KUKA KRL program: MyProgram_015().src

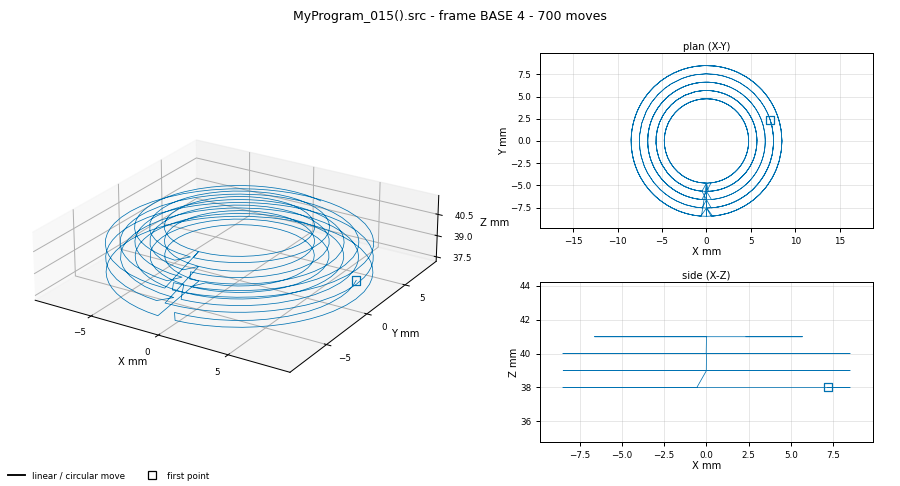
[picture p0: tool path of MyProgram_015().src in frame BASE 4, 700 of 700 moves have a stored position in this frame; points joined in program order, loops and branches not executed]
&ACCESS RVP
&REL 1
&PARAM TEMPLATE = C:\KRC\Roboter\Template\vorgabe
&PARAM EDITMASK = *
DEF MyProgram_015()
; ---- Setting reference (Base) ----
$BASE = BASE_DATA[4]

; --------------------------
; ---- Setting tool (TCP) ----
$TOOL = TOOL_DATA[3]
; --------------------------

$VEL.CP = VEL_APROX_PRINT
Startdeposition()
$VEL.CP = VEL_PRINT
LIN {X 7.1653,Y 2.4052,Z 38,A -2.3243,B 0,C 0,E1 0.1598,E2 90.0714} C_DIS
LIN {X 7.3844,Y 1.6056,Z 38,A -2.3508,B 0,C 0,E1 0.1598,E2 90.0719} C_DIS
LIN {X 7.5274,Y 0.6858,Z 38,A -2.3849,B 0,C 0,E1 0.1598,E2 90.0719} C_DIS
LIN {X 7.5543,Y -0.2016,Z 38,A -2.4217,B 0,C 0,E1 0.1598,E2 90.0719} C_DIS
LIN {X 7.4214,Y -1.405,Z 38,A -2.4775,B 0,C 0,E1 0.1598,E2 90.0714} C_DIS
LIN {X 7.2331,Y -2.1884,Z 38,A -2.5182,B 0,C 0,E1 0.1598,E2 90.0717} C_DIS
LIN {X 6.879,Y -3.1316,Z 38,A -2.5714,B 0,C 0,E1 0.1598,E2 90.0717} C_DIS
LIN {X 6.1912,Y -4.3324,Z 38,A -2.6476,B 0,C 0,E1 0.1598,E2 90.0712} C_DIS
LIN {X 5.3371,Y -5.3523,Z 38,A -2.7227,B 0,C 0,E1 0.1598,E2 90.0714} C_DIS
LIN {X 4.6683,Y -5.9424,Z 38,A -2.7727,B 0,C 0,E1 0.1598,E2 90.0717} C_DIS
LIN {X 3.7573,Y -6.5524,Z 38,A -2.8321,B 0,C 0,E1 0.1598,E2 90.0717} C_DIS
LIN {X 2.7191,Y -7.0514,Z 38,A -2.8915,B 0,C 0,E1 0.1598,E2 90.0717} C_DIS
LIN {X 1.7846,Y -7.3382,Z 38,A -2.9381,B 0,C 0,E1 0.1598,E2 90.0717} C_DIS
LIN {X 1.0166,Y -7.4849,Z 38,A -2.9725,B 0,C 0,E1 0.1598,E2 90.0717} C_DIS
LIN {X 0.0417,Y -7.5527,Z 38,A -3.0111,B 0,C 0,E1 0.1598,E2 90.0716} C_DIS
Enddeposition()
LIN {X 0.0417,Y -7.5527,Z 38,A -3.0111,B 0,C 0,E1 0.1598,E2 90.0716} C_DIS
Startdeposition()
$VEL.CP = VEL_PRINT
LIN {X 0.6842,Y -8.4602,Z 38,A -3.0258,B 0,C 0,E1 0.1598,E2 90.071} C_DIS
LIN {X 1.5115,Y -8.3518,Z 38,A -2.9914,B 0,C 0,E1 0.1598,E2 90.0716} C_DIS
LIN {X 2.525,Y -8.1061,Z 38,A -2.9438,B 0,C 0,E1 0.1598,E2 90.0716} C_DIS
LIN {X 3.5839,Y -7.6978,Z 38,A -2.8876,B 0,C 0,E1 0.1598,E2 90.0716} C_DIS
LIN {X 4.65,Y -7.0996,Z 38,A -2.8229,B 0,C 0,E1 0.1598,E2 90.0716} C_DIS
LIN {X 5.3529,Y -6.5853,Z 38,A -2.7752,B 0,C 0,E1 0.1598,E2 90.0717} C_DIS
LIN {X 5.9995,Y -6.0018,Z 38,A -2.7266,B 0,C 0,E1 0.1598,E2 90.0717} C_DIS
LIN {X 6.5829,Y -5.3553,Z 38,A -2.6775,B 0,C 0,E1 0.1598,E2 90.0717} C_DIS
LIN {X 7.0969,Y -4.6523,Z 38,A -2.6286,B 0,C 0,E1 0.1598,E2 90.0718} C_DIS
LIN {X 7.5367,Y -3.9006,Z 38,A -2.5804,B 0,C 0,E1 0.1598,E2 90.0718} C_DIS
LIN {X 7.8972,Y -3.1077,Z 38,A -2.5332,B 0,C 0,E1 0.1598,E2 90.0718} C_DIS
LIN {X 8.1746,Y -2.2821,Z 38,A -2.4878,B 0,C 0,E1 0.1598,E2 90.0718} C_DIS
LIN {X 8.4206,Y -1.0958,Z 38,A -2.4277,B 0,C 0,E1 0.1598,E2 90.0716} C_DIS
LIN {X 8.4922,Y -0.0069,Z 38,A -2.3787,B 0,C 0,E1 0.1598,E2 90.0717} C_DIS
LIN {X 8.4074,Y 1.1944,Z 38,A -2.3304,B 0,C 0,E1 0.1598,E2 90.0717} C_DIS
LIN {X 8.161,Y 2.3308,Z 38,A -2.291,B 0,C 0,E1 0.1598,E2 90.0717} C_DIS
LIN {X 7.8787,Y 3.1561,Z 38,A -2.2666,B 0,C 0,E1 0.1598,E2 90.0721} C_DIS
LIN {X 7.5129,Y 3.9479,Z 38,A -2.2464,B 0,C 0,E1 0.1598,E2 90.0721} C_DIS
LIN {X 7.0677,Y 4.698,Z 38,A -2.2309,B 0,C 0,E1 0.1598,E2 90.0723} C_DIS
LIN {X 6.5481,Y 5.3986,Z 38,A -2.2203,B 0,C 0,E1 0.1598,E2 90.0723} C_DIS
LIN {X 5.9597,Y 6.0425,Z 38,A -2.2146,B 0,C 0,E1 0.1598,E2 90.0723} C_DIS
LIN {X 4.9857,Y 6.8745,Z 38,A -2.215,B 0,C 0,E1 0.1598,E2 90.0723} C_DIS
LIN {X 3.9863,Y 7.4937,Z 38,A -2.2257,B 0,C 0,E1 0.1598,E2 90.0723} C_DIS
LIN {X 3.2149,Y 7.8556,Z 38,A -2.239,B 0,C 0,E1 0.1598,E2 90.0725} C_DIS
LIN {X 2.411,Y 8.1383,Z 38,A -2.2567,B 0,C 0,E1 0.1598,E2 90.0725} C_DIS
LIN {X 1.5828,Y 8.3389,Z 38,A -2.2788,B 0,C 0,E1 0.1598,E2 90.0725} C_DIS
LIN {X 0.7387,Y 8.4557,Z 38,A -2.3051,B 0,C 0,E1 0.1598,E2 90.0725} C_DIS
LIN {X -0.4396,Y 8.4801,Z 38,A -2.3475,B 0,C 0,E1 0.1598,E2 90.0725} C_DIS
LIN {X -1.5024,Y 8.3537,Z 38,A -2.3921,B 0,C 0,E1 0.1598,E2 90.0724} C_DIS
LIN {X -2.5423,Y 8.1007,Z 38,A -2.4412,B 0,C 0,E1 0.1598,E2 90.0723} C_DIS
LIN {X -3.7176,Y 7.6272,Z 38,A -2.5045,B 0,C 0,E1 0.1598,E2 90.0721} C_DIS
LIN {X -4.4451,Y 7.2274,Z 38,A -2.5483,B 0,C 0,E1 0.1598,E2 90.0721} C_DIS
LIN {X -5.1302,Y 6.7585,Z 38,A -2.5934,B 0,C 0,E1 0.1598,E2 90.0721} C_DIS
LIN {X -5.7662,Y 6.2249,Z 38,A -2.6394,B 0,C 0,E1 0.1598,E2 90.0719} C_DIS
LIN {X -6.3472,Y 5.6318,Z 38,A -2.6858,B 0,C 0,E1 0.1598,E2 90.0719} C_DIS
LIN {X -6.8675,Y 4.9849,Z 38,A -2.7323,B 0,C 0,E1 0.1598,E2 90.0717} C_DIS
LIN {X -7.3221,Y 4.2902,Z 38,A -2.7784,B 0,C 0,E1 0.1598,E2 90.0717} C_DIS
LIN {X -7.7067,Y 3.5544,Z 38,A -2.8236,B 0,C 0,E1 0.1598,E2 90.0715} C_DIS
LIN {X -8.0173,Y 2.7844,Z 38,A -2.8675,B 0,C 0,E1 0.1598,E2 90.0715} C_DIS
LIN {X -8.2508,Y 1.9876,Z 38,A -2.9098,B 0,C 0,E1 0.1598,E2 90.0714} C_DIS
LIN {X -8.405,Y 1.1717,Z 38,A -2.9499,B 0,C 0,E1 0.1598,E2 90.0713} C_DIS
LIN {X -8.4896,Y 0.1374,Z 38,A -2.9964,B 0,C 0,E1 0.1598,E2 90.0709} C_DIS
LIN {X -8.4227,Y -1.0517,Z 38,A -3.0441,B 0,C 0,E1 0.1598,E2 90.0708} C_DIS
LIN {X -8.2776,Y -1.875,Z 38,A -3.0739,B 0,C 0,E1 0.1598,E2 90.0711} C_DIS
LIN {X -8.0525,Y -2.6802,Z 38,A -3.0997,B 0,C 0,E1 0.1598,E2 90.0711} C_DIS
LIN {X -7.7494,Y -3.4593,Z 38,A -3.1216,B 0,C 0,E1 0.1598,E2 90.0711} C_DIS
LIN {X -7.371,Y -4.2047,Z 38,A -3.1392,B 0,C 0,E1 0.1598,E2 90.0711} C_DIS
LIN {X -6.9212,Y -4.9093,Z 38,A -3.1526,B 0,C 0,E1 0.1598,E2 90.0711} C_DIS
LIN {X -6.4044,Y -5.5663,Z 38,A -3.1615,B 0,C 0,E1 0.1598,E2 90.0711} C_DIS
LIN {X -5.8257,Y -6.1694,Z 38,A -3.1658,B 0,C 0,E1 0.1598,E2 90.0711} C_DIS
LIN {X -5.1905,Y -6.7127,Z 38,A -3.1656,B 0,C 0,E1 0.1598,E2 90.0711} C_DIS
LIN {X -4.5049,Y -7.1909,Z 38,A -3.1608,B 0,C 0,E1 0.1598,E2 90.0712} C_DIS
LIN {X -3.7757,Y -7.5993,Z 38,A -3.1514,B 0,C 0,E1 0.1598,E2 90.0712} C_DIS
LIN {X -3.0099,Y -7.9343,Z 38,A -3.1376,B 0,C 0,E1 0.1598,E2 90.0713} C_DIS
LIN {X -2.2145,Y -8.1913,Z 38,A -3.1194,B 0,C 0,E1 0.1598,E2 90.0713} C_DIS
LIN {X -1.3979,Y -8.3693,Z 38,A -3.0971,B 0,C 0,E1 0.1598,E2 90.0714} C_DIS
LIN {X -0.5677,Y -8.4665,Z 38,A -3.0708,B 0,C 0,E1 0.1598,E2 90.0714} C_DIS
LIN {X -0.5677,Y -8.4665,Z 38,A -3.0708,B 0,C 0,E1 0.1598,E2 90.0714} C_DIS
Enddeposition()
LIN {X 0.0009,Y -4.7541,Z 39,A -2.8773,B 0,C 0,E1 0.1598,E2 90.0604} C_DIS
Startdeposition()
$VEL.CP = VEL_PRINT
LIN {X 0.0009,Y -4.7541,Z 39,A -2.8831,B 0,C 0,E1 0.1598,E2 90.0661} C_DIS
LIN {X -0.8426,Y -4.6756,Z 39,A -2.9156,B 0,C 0,E1 0.1598,E2 90.071} C_DIS
LIN {X -1.4993,Y -4.5079,Z 39,A -2.9332,B 0,C 0,E1 0.1598,E2 90.0716} C_DIS
LIN {X -2.2007,Y -4.2093,Z 39,A -2.9463,B 0,C 0,E1 0.1598,E2 90.0716} C_DIS
LIN {X -2.7089,Y -3.9031,Z 39,A -2.9519,B 0,C 0,E1 0.1598,E2 90.0716} C_DIS
LIN {X -3.2362,Y -3.4772,Z 39,A -2.9532,B 0,C 0,E1 0.1598,E2 90.0716} C_DIS
LIN {X -3.6987,Y -2.9818,Z 39,A -2.9491,B 0,C 0,E1 0.1598,E2 90.0716} C_DIS
LIN {X -4.0854,Y -2.4248,Z 39,A -2.9397,B 0,C 0,E1 0.1598,E2 90.0715} C_DIS
LIN {X -4.3899,Y -1.8192,Z 39,A -2.9251,B 0,C 0,E1 0.1598,E2 90.0715} C_DIS
LIN {X -4.6019,Y -1.1753,Z 39,A -2.9056,B 0,C 0,E1 0.1598,E2 90.0715} C_DIS
LIN {X -4.7232,Y -0.5085,Z 39,A -2.8818,B 0,C 0,E1 0.1598,E2 90.0715} C_DIS
LIN {X -4.7486,Y 0.1689,Z 39,A -2.8541,B 0,C 0,E1 0.1598,E2 90.0715} C_DIS
LIN {X -4.6757,Y 0.8428,Z 39,A -2.8228,B 0,C 0,E1 0.1598,E2 90.0715} C_DIS
LIN {X -4.508,Y 1.4995,Z 39,A -2.7889,B 0,C 0,E1 0.1598,E2 90.0716} C_DIS
LIN {X -4.2489,Y 2.1259,Z 39,A -2.7528,B 0,C 0,E1 0.1598,E2 90.0716} C_DIS
LIN {X -3.8529,Y 2.7772,Z 39,A -2.7106,B 0,C 0,E1 0.1598,E2 90.0717} C_DIS
LIN {X -3.4771,Y 3.2361,Z 39,A -2.6774,B 0,C 0,E1 0.1598,E2 90.0719} C_DIS
LIN {X -2.9816,Y 3.6987,Z 39,A -2.6396,B 0,C 0,E1 0.1598,E2 90.0719} C_DIS
LIN {X -2.4252,Y 4.0858,Z 39,A -2.6027,B 0,C 0,E1 0.1598,E2 90.072} C_DIS
LIN {X -1.8189,Y 4.3894,Z 39,A -2.5676,B 0,C 0,E1 0.1598,E2 90.0721} C_DIS
LIN {X -1.1762,Y 4.6049,Z 39,A -2.5348,B 0,C 0,E1 0.1598,E2 90.0721} C_DIS
LIN {X -0.5089,Y 4.7255,Z 39,A -2.5051,B 0,C 0,E1 0.1598,E2 90.0722} C_DIS
LIN {X 0.1687,Y 4.7484,Z 39,A -2.4791,B 0,C 0,E1 0.1598,E2 90.0722} C_DIS
LIN {X 0.8425,Y 4.6752,Z 39,A -2.4574,B 0,C 0,E1 0.1598,E2 90.0722} C_DIS
LIN {X 1.5,Y 4.5099,Z 39,A -2.4402,B 0,C 0,E1 0.1598,E2 90.0722} C_DIS
LIN {X 2.2007,Y 4.2093,Z 39,A -2.4271,B 0,C 0,E1 0.1598,E2 90.0722} C_DIS
LIN {X 2.7772,Y 3.8529,Z 39,A -2.4209,B 0,C 0,E1 0.1598,E2 90.0722} C_DIS
LIN {X 3.2376,Y 3.4785,Z 39,A -2.4199,B 0,C 0,E1 0.1598,E2 90.0722} C_DIS
LIN {X 3.6983,Y 2.9813,Z 39,A -2.424,B 0,C 0,E1 0.1598,E2 90.0722} C_DIS
LIN {X 4.0856,Y 2.425,Z 39,A -2.4333,B 0,C 0,E1 0.1598,E2 90.0722} C_DIS
LIN {X 4.3905,Y 1.8194,Z 39,A -2.4479,B 0,C 0,E1 0.1598,E2 90.0721} C_DIS
LIN {X 4.6049,Y 1.1762,Z 39,A -2.4673,B 0,C 0,E1 0.1598,E2 90.0721} C_DIS
LIN {X 4.7256,Y 0.5089,Z 39,A -2.4913,B 0,C 0,E1 0.1598,E2 90.072} C_DIS
LIN {X 4.7479,Y -0.1687,Z 39,A -2.5193,B 0,C 0,E1 0.1598,E2 90.072} C_DIS
LIN {X 4.6756,Y -0.8426,Z 39,A -2.5506,B 0,C 0,E1 0.1598,E2 90.072} C_DIS
LIN {X 4.5077,Y -1.4992,Z 39,A -2.5848,B 0,C 0,E1 0.1598,E2 90.0719} C_DIS
LIN {X 4.2489,Y -2.1257,Z 39,A -2.621,B 0,C 0,E1 0.1598,E2 90.0719} C_DIS
LIN {X 3.9047,Y -2.7098,Z 39,A -2.6585,B 0,C 0,E1 0.1598,E2 90.0719} C_DIS
LIN {X 3.4774,Y -3.2362,Z 39,A -2.6967,B 0,C 0,E1 0.1598,E2 90.0719} C_DIS
LIN {X 2.9809,Y -3.6975,Z 39,A -2.7346,B 0,C 0,E1 0.1598,E2 90.0719} C_DIS
LIN {X 2.4243,Y -4.0842,Z 39,A -2.7715,B 0,C 0,E1 0.1598,E2 90.0719} C_DIS
LIN {X 1.8189,Y -4.3891,Z 39,A -2.8068,B 0,C 0,E1 0.1598,E2 90.0718} C_DIS
LIN {X 1.176,Y -4.6047,Z 39,A -2.8396,B 0,C 0,E1 0.1598,E2 90.0718} C_DIS
LIN {X 0.5089,Y -4.7255,Z 39,A -2.8692,B 0,C 0,E1 0.1598,E2 90.0718} C_DIS
LIN {X 0.5089,Y -4.7255,Z 39,A -2.8692,B 0,C 0,E1 0.1598,E2 90.0718} C_DIS
Enddeposition()
LIN {X 0.0121,Y -5.6872,Z 39,A -2.9273,B 0,C 0,E1 0.1598,E2 90.0705} C_DIS
Startdeposition()
$VEL.CP = VEL_PRINT
LIN {X 0.6271,Y -5.648,Z 39,A -2.9042,B 0,C 0,E1 0.1598,E2 90.0716} C_DIS
LIN {X 1.4348,Y -5.4997,Z 39,A -2.8683,B 0,C 0,E1 0.1598,E2 90.0717} C_DIS
LIN {X 2.2127,Y -5.2362,Z 39,A -2.8285,B 0,C 0,E1 0.1598,E2 90.0717} C_DIS
LIN {X 2.945,Y -4.8639,Z 39,A -2.7857,B 0,C 0,E1 0.1598,E2 90.0717} C_DIS
LIN {X 3.6144,Y -4.3879,Z 39,A -2.7408,B 0,C 0,E1 0.1598,E2 90.0718} C_DIS
LIN {X 4.4069,Y -3.6004,Z 39,A -2.678,B 0,C 0,E1 0.1598,E2 90.0718} C_DIS
LIN {X 4.9608,Y -2.7789,Z 39,A -2.6226,B 0,C 0,E1 0.1598,E2 90.0718} C_DIS
LIN {X 5.3715,Y -1.8773,Z 39,A -2.5689,B 0,C 0,E1 0.1598,E2 90.0716} C_DIS
LIN {X 5.6395,Y -0.7198,Z 39,A -2.5095,B 0,C 0,E1 0.1598,E2 90.0715} C_DIS
LIN {X 5.6848,Y 0.1071,Z 39,A -2.4729,B 0,C 0,E1 0.1598,E2 90.0719} C_DIS
LIN {X 5.6086,Y 0.9317,Z 39,A -2.4406,B 0,C 0,E1 0.1598,E2 90.0719} C_DIS
LIN {X 5.4132,Y 1.7365,Z 39,A -2.4136,B 0,C 0,E1 0.1598,E2 90.0719} C_DIS
LIN {X 5.1041,Y 2.5047,Z 39,A -2.3923,B 0,C 0,E1 0.1598,E2 90.072} C_DIS
LIN {X 4.6855,Y 3.2194,Z 39,A -2.3773,B 0,C 0,E1 0.1598,E2 90.072} C_DIS
LIN {X 4.1689,Y 3.8668,Z 39,A -2.3689,B 0,C 0,E1 0.1598,E2 90.0722} C_DIS
LIN {X 3.562,Y 4.4302,Z 39,A -2.3673,B 0,C 0,E1 0.1598,E2 90.0722} C_DIS
LIN {X 2.8807,Y 4.9007,Z 39,A -2.3725,B 0,C 0,E1 0.1598,E2 90.0722} C_DIS
LIN {X 2.1386,Y 5.2681,Z 39,A -2.3843,B 0,C 0,E1 0.1598,E2 90.0723} C_DIS
LIN {X 1.3506,Y 5.5226,Z 39,A -2.4026,B 0,C 0,E1 0.1598,E2 90.0723} C_DIS
LIN {X 0.534,Y 5.6605,Z 39,A -2.4269,B 0,C 0,E1 0.1598,E2 90.0723} C_DIS
LIN {X -0.2939,Y 5.6768,Z 39,A -2.4567,B 0,C 0,E1 0.1598,E2 90.0723} C_DIS
LIN {X -1.3193,Y 5.5356,Z 39,A -2.5005,B 0,C 0,E1 0.1598,E2 90.0723} C_DIS
LIN {X -2.4585,Y 5.1308,Z 39,A -2.5596,B 0,C 0,E1 0.1598,E2 90.0721} C_DIS
LIN {X -3.3251,Y 4.6118,Z 39,A -2.6135,B 0,C 0,E1 0.1598,E2 90.072} C_DIS
LIN {X -3.9455,Y 4.0938,Z 39,A -2.6583,B 0,C 0,E1 0.1598,E2 90.0719} C_DIS
LIN {X -4.4848,Y 3.4918,Z 39,A -2.7036,B 0,C 0,E1 0.1598,E2 90.0718} C_DIS
LIN {X -4.9332,Y 2.8198,Z 39,A -2.7485,B 0,C 0,E1 0.1598,E2 90.0717} C_DIS
LIN {X -5.2834,Y 2.0919,Z 39,A -2.7921,B 0,C 0,E1 0.1598,E2 90.0716} C_DIS
LIN {X -5.5269,Y 1.3217,Z 39,A -2.8337,B 0,C 0,E1 0.1598,E2 90.0715} C_DIS
LIN {X -5.661,Y 0.5248,Z 39,A -2.8723,B 0,C 0,E1 0.1598,E2 90.0715} C_DIS
LIN {X -5.6768,Y -0.283,Z 39,A -2.907,B 0,C 0,E1 0.1598,E2 90.0714} C_DIS
LIN {X -5.5777,Y -1.0848,Z 39,A -2.9374,B 0,C 0,E1 0.1598,E2 90.0714} C_DIS
LIN {X -5.3693,Y -1.8654,Z 39,A -2.9628,B 0,C 0,E1 0.1598,E2 90.0713} C_DIS
LIN {X -5.0517,Y -2.6086,Z 39,A -2.9826,B 0,C 0,E1 0.1598,E2 90.0713} C_DIS
LIN {X -4.3493,Y -3.6677,Z 39,A -3.0014,B 0,C 0,E1 0.1598,E2 90.071} C_DIS
LIN {X -3.8838,Y -4.1512,Z 39,A -3.0052,B 0,C 0,E1 0.1598,E2 90.0714} C_DIS
LIN {X -3.2642,Y -4.6597,Z 39,A -3.004,B 0,C 0,E1 0.1598,E2 90.0714} C_DIS
LIN {X -2.5122,Y -5.0989,Z 39,A -2.9952,B 0,C 0,E1 0.1598,E2 90.0714} C_DIS
LIN {X -1.8695,Y -5.3681,Z 39,A -2.9831,B 0,C 0,E1 0.1598,E2 90.0716} C_DIS
LIN {X -1.1992,Y -5.5587,Z 39,A -2.9666,B 0,C 0,E1 0.1598,E2 90.0716} C_DIS
LIN {X -0.51,Y -5.6605,Z 39,A -2.9457,B 0,C 0,E1 0.1598,E2 90.0716} C_DIS
LIN {X -0.51,Y -5.6605,Z 39,A -2.9457,B 0,C 0,E1 0.1598,E2 90.0716} C_DIS
Enddeposition()
LIN {X 0.0069,Y -6.6201,Z 39,A -2.9665,B 0,C 0,E1 0.1598,E2 90.0704} C_DIS
Startdeposition()
$VEL.CP = VEL_PRINT
LIN {X -0.8789,Y -6.5615,Z 39,A -2.9976,B 0,C 0,E1 0.1598,E2 90.0715} C_DIS
LIN {X -1.5766,Y -6.4282,Z 39,A -3.0176,B 0,C 0,E1 0.1598,E2 90.0715} C_DIS
LIN {X -2.2562,Y -6.2214,Z 39,A -3.0337,B 0,C 0,E1 0.1598,E2 90.0715} C_DIS
LIN {X -2.9104,Y -5.9449,Z 39,A -3.0459,B 0,C 0,E1 0.1598,E2 90.0715} C_DIS
LIN {X -3.5318,Y -5.6008,Z 39,A -3.0541,B 0,C 0,E1 0.1598,E2 90.0715} C_DIS
LIN {X -4.1104,Y -5.1886,Z 39,A -3.0578,B 0,C 0,E1 0.1598,E2 90.0715} C_DIS
LIN {X -4.6423,Y -4.7178,Z 39,A -3.0573,B 0,C 0,E1 0.1598,E2 90.0714} C_DIS
LIN {X -5.1209,Y -4.193,Z 39,A -3.0526,B 0,C 0,E1 0.1598,E2 90.0714} C_DIS
LIN {X -5.5416,Y -3.6206,Z 39,A -3.0438,B 0,C 0,E1 0.1598,E2 90.0714} C_DIS
LIN {X -5.8984,Y -3.0063,Z 39,A -3.0308,B 0,C 0,E1 0.1598,E2 90.0714} C_DIS
LIN {X -6.3003,Y -2.0434,Z 39,A -3.0045,B 0,C 0,E1 0.1598,E2 90.0711} C_DIS
LIN {X -6.5074,Y -1.2136,Z 39,A -2.9772,B 0,C 0,E1 0.1598,E2 90.0713} C_DIS
LIN {X -6.5996,Y -0.5358,Z 39,A -2.952,B 0,C 0,E1 0.1598,E2 90.0713} C_DIS
LIN {X -6.6169,Y 0.1481,Z 39,A -2.9237,B 0,C 0,E1 0.1598,E2 90.0714} C_DIS
LIN {X -6.5679,Y 0.8304,Z 39,A -2.893,B 0,C 0,E1 0.1598,E2 90.0714} C_DIS
LIN {X -6.4473,Y 1.5038,Z 39,A -2.8601,B 0,C 0,E1 0.1598,E2 90.0715} C_DIS
LIN {X -6.2582,Y 2.1612,Z 39,A -2.8253,B 0,C 0,E1 0.1598,E2 90.0715} C_DIS
LIN {X -6.0017,Y 2.7955,Z 39,A -2.789,B 0,C 0,E1 0.1598,E2 90.0716} C_DIS
LIN {X -5.5005,Y 3.6898,Z 39,A -2.7326,B 0,C 0,E1 0.1598,E2 90.0716} C_DIS
LIN {X -4.946,Y 4.3986,Z 39,A -2.6823,B 0,C 0,E1 0.1598,E2 90.0718} C_DIS
LIN {X -4.4392,Y 4.91,Z 39,A -2.6421,B 0,C 0,E1 0.1598,E2 90.0719} C_DIS
LIN {X -3.88,Y 5.3634,Z 39,A -2.6023,B 0,C 0,E1 0.1598,E2 90.0719} C_DIS
LIN {X -3.2751,Y 5.7537,Z 39,A -2.5635,B 0,C 0,E1 0.1598,E2 90.0721} C_DIS
LIN {X -2.6302,Y 6.0739,Z 39,A -2.5262,B 0,C 0,E1 0.1598,E2 90.0721} C_DIS
LIN {X -1.9552,Y 6.3238,Z 39,A -2.4907,B 0,C 0,E1 0.1598,E2 90.0722} C_DIS
LIN {X -1.257,Y 6.4989,Z 39,A -2.4576,B 0,C 0,E1 0.1598,E2 90.0722} C_DIS
LIN {X -0.5439,Y 6.5973,Z 39,A -2.4271,B 0,C 0,E1 0.1598,E2 90.0723} C_DIS
LIN {X 0.1756,Y 6.6151,Z 39,A -2.3998,B 0,C 0,E1 0.1598,E2 90.0723} C_DIS
LIN {X 0.8933,Y 6.5597,Z 39,A -2.3757,B 0,C 0,E1 0.1598,E2 90.0723} C_DIS
LIN {X 1.9111,Y 6.3417,Z 39,A -2.3473,B 0,C 0,E1 0.1598,E2 90.0724} C_DIS
LIN {X 2.7735,Y 6.0107,Z 39,A -2.3296,B 0,C 0,E1 0.1598,E2 90.0724} C_DIS
LIN {X 3.4259,Y 5.6639,Z 39,A -2.3202,B 0,C 0,E1 0.1598,E2 90.0724} C_DIS
LIN {X 4.0365,Y 5.2479,Z 39,A -2.3153,B 0,C 0,E1 0.1598,E2 90.0724} C_DIS
LIN {X 4.5943,Y 4.7632,Z 39,A -2.3153,B 0,C 0,E1 0.1598,E2 90.0724} C_DIS
LIN {X 5.0973,Y 4.2221,Z 39,A -2.3198,B 0,C 0,E1 0.1598,E2 90.0723} C_DIS
LIN {X 5.5358,Y 3.6275,Z 39,A -2.3289,B 0,C 0,E1 0.1598,E2 90.0723} C_DIS
LIN {X 5.9075,Y 2.989,Z 39,A -2.3424,B 0,C 0,E1 0.1598,E2 90.0723} C_DIS
LIN {X 6.2011,Y 2.3111,Z 39,A -2.3604,B 0,C 0,E1 0.1598,E2 90.0722} C_DIS
LIN {X 6.4207,Y 1.6057,Z 39,A -2.3823,B 0,C 0,E1 0.1598,E2 90.0722} C_DIS
LIN {X 6.559,Y 0.88,Z 39,A -2.4081,B 0,C 0,E1 0.1598,E2 90.0721} C_DIS
LIN {X 6.6176,Y 0.1435,Z 39,A -2.4374,B 0,C 0,E1 0.1598,E2 90.0721} C_DIS
LIN {X 6.5909,Y -0.5948,Z 39,A -2.4698,B 0,C 0,E1 0.1598,E2 90.072} C_DIS
LIN {X 6.484,Y -1.3258,Z 39,A -2.5049,B 0,C 0,E1 0.1598,E2 90.072} C_DIS
LIN {X 6.2975,Y -2.0407,Z 39,A -2.5423,B 0,C 0,E1 0.1598,E2 90.0719} C_DIS
LIN {X 6.0302,Y -2.7295,Z 39,A -2.5815,B 0,C 0,E1 0.1598,E2 90.0719} C_DIS
LIN {X 5.6894,Y -3.3851,Z 39,A -2.622,B 0,C 0,E1 0.1598,E2 90.0719} C_DIS
LIN {X 5.2768,Y -3.9982,Z 39,A -2.6633,B 0,C 0,E1 0.1598,E2 90.0719} C_DIS
LIN {X 4.7988,Y -4.5617,Z 39,A -2.7049,B 0,C 0,E1 0.1598,E2 90.0719} C_DIS
LIN {X 4.2592,Y -5.0666,Z 39,A -2.7462,B 0,C 0,E1 0.1598,E2 90.0718} C_DIS
LIN {X 3.6677,Y -5.5093,Z 39,A -2.7868,B 0,C 0,E1 0.1598,E2 90.0718} C_DIS
LIN {X 3.031,Y -5.8841,Z 39,A -2.8262,B 0,C 0,E1 0.1598,E2 90.0718} C_DIS
LIN {X 2.356,Y -6.1843,Z 39,A -2.8638,B 0,C 0,E1 0.1598,E2 90.0718} C_DIS
LIN {X 1.6522,Y -6.409,Z 39,A -2.8992,B 0,C 0,E1 0.1598,E2 90.0717} C_DIS
LIN {X 0.9278,Y -6.5543,Z 39,A -2.9319,B 0,C 0,E1 0.1598,E2 90.0717} C_DIS
LIN {X 0.0069,Y -6.6201,Z 39,A -2.9685,B 0,C 0,E1 0.1598,E2 90.0717} C_DIS
Enddeposition()
LIN {X 0.0069,Y -6.6201,Z 39,A -2.9685,B 0,C 0,E1 0.1598,E2 90.0717} C_DIS
Startdeposition()
$VEL.CP = VEL_PRINT
LIN {X 0.5273,Y -7.5341,Z 39,A -2.9879,B 0,C 0,E1 0.1598,E2 90.071} C_DIS
LIN {X 1.2198,Y -7.4551,Z 39,A -2.9597,B 0,C 0,E1 0.1598,E2 90.0716} C_DIS
LIN {X 1.9017,Y -7.3109,Z 39,A -2.9286,B 0,C 0,E1 0.1598,E2 90.0716} C_DIS
LIN {X 2.732,Y -7.0467,Z 39,A -2.8869,B 0,C 0,E1 0.1598,E2 90.0716} C_DIS
LIN {X 3.6901,Y -6.5944,Z 39,A -2.8324,B 0,C 0,E1 0.1598,E2 90.0717} C_DIS
LIN {X 4.5143,Y -6.0548,Z 39,A -2.7791,B 0,C 0,E1 0.1598,E2 90.0717} C_DIS
LIN {X 5.1213,Y -5.5521,Z 39,A -2.7354,B 0,C 0,E1 0.1598,E2 90.0717} C_DIS
LIN {X 5.8029,Y -4.8409,Z 39,A -2.6799,B 0,C 0,E1 0.1598,E2 90.0717} C_DIS
LIN {X 6.5456,Y -3.7767,Z 39,A -2.6069,B 0,C 0,E1 0.1598,E2 90.0714} C_DIS
LIN {X 7.0796,Y -2.6425,Z 39,A -2.5387,B 0,C 0,E1 0.1598,E2 90.0714} C_DIS
LIN {X 7.4028,Y -1.5014,Z 39,A -2.4782,B 0,C 0,E1 0.1598,E2 90.0714} C_DIS
LIN {X 7.5505,Y -0.3487,Z 39,A -2.4237,B 0,C 0,E1 0.1598,E2 90.0716} C_DIS
LIN {X 7.5342,Y 0.5909,Z 39,A -2.3844,B 0,C 0,E1 0.1598,E2 90.0719} C_DIS
LIN {X 7.3598,Y 1.6941,Z 39,A -2.3436,B 0,C 0,E1 0.1598,E2 90.0717} C_DIS
LIN {X 7.149,Y 2.4398,Z 39,A -2.3199,B 0,C 0,E1 0.1598,E2 90.0721} C_DIS
LIN {X 6.8615,Y 3.1595,Z 39,A -2.2999,B 0,C 0,E1 0.1598,E2 90.0721} C_DIS
LIN {X 6.501,Y 3.8455,Z 39,A -2.2839,B 0,C 0,E1 0.1598,E2 90.0722} C_DIS
LIN {X 6.0727,Y 4.4914,Z 39,A -2.2723,B 0,C 0,E1 0.1598,E2 90.0722} C_DIS
LIN {X 5.3507,Y 5.3387,Z 39,A -2.2627,B 0,C 0,E1 0.1598,E2 90.0722} C_DIS
LIN {X 4.6598,Y 5.9456,Z 39,A -2.2625,B 0,C 0,E1 0.1598,E2 90.0723} C_DIS
LIN {X 3.7396,Y 6.5672,Z 39,A -2.27,B 0,C 0,E1 0.1598,E2 90.0723} C_DIS
LIN {X 2.8216,Y 7.0046,Z 39,A -2.2854,B 0,C 0,E1 0.1598,E2 90.0723} C_DIS
LIN {X 2.0525,Y 7.2694,Z 39,A -2.3026,B 0,C 0,E1 0.1598,E2 90.0724} C_DIS
LIN {X 0.9279,Y 7.5,Z 39,A -2.3344,B 0,C 0,E1 0.1598,E2 90.0724} C_DIS
LIN {X -0.0433,Y 7.5579,Z 39,A -2.3678,B 0,C 0,E1 0.1598,E2 90.0724} C_DIS
LIN {X -1.2589,Y 7.4475,Z 39,A -2.4173,B 0,C 0,E1 0.1598,E2 90.0724} C_DIS
LIN {X -2.0232,Y 7.2762,Z 39,A -2.4528,B 0,C 0,E1 0.1598,E2 90.0723} C_DIS
LIN {X -2.7658,Y 7.0275,Z 39,A -2.4907,B 0,C 0,E1 0.1598,E2 90.0723} C_DIS
LIN {X -3.9527,Y 6.4403,Z 39,A -2.5592,B 0,C 0,E1 0.1598,E2 90.072} C_DIS
LIN {X -4.6822,Y 5.9317,Z 39,A -2.6077,B 0,C 0,E1 0.1598,E2 90.072} C_DIS
LIN {X -5.4823,Y 5.2003,Z 39,A -2.668,B 0,C 0,E1 0.1598,E2 90.0717} C_DIS
LIN {X -6.1876,Y 4.3377,Z 39,A -2.7303,B 0,C 0,E1 0.1598,E2 90.0716} C_DIS
LIN {X -6.777,Y 3.3429,Z 39,A -2.794,B 0,C 0,E1 0.1598,E2 90.0714} C_DIS
LIN {X -7.2899,Y 1.9923,Z 39,A -2.8695,B 0,C 0,E1 0.1598,E2 90.0708} C_DIS
LIN {X -7.5202,Y 0.7015,Z 39,A -2.9326,B 0,C 0,E1 0.1598,E2 90.0708} C_DIS
LIN {X -7.5526,Y -0.1159,Z 39,A -2.9688,B 0,C 0,E1 0.1598,E2 90.0712} C_DIS
LIN {X -7.4936,Y -0.9318,Z 39,A -3.0012,B 0,C 0,E1 0.1598,E2 90.0712} C_DIS
LIN {X -7.351,Y -1.7371,Z 39,A -3.03,B 0,C 0,E1 0.1598,E2 90.0712} C_DIS
LIN {X -7.0047,Y -2.8377,Z 39,A -3.0636,B 0,C 0,E1 0.1598,E2 90.0709} C_DIS
LIN {X -6.6345,Y -3.6173,Z 39,A -3.0833,B 0,C 0,E1 0.1598,E2 90.0712} C_DIS
LIN {X -5.9557,Y -4.651,Z 39,A -3.1019,B 0,C 0,E1 0.1598,E2 90.0708} C_DIS
LIN {X -5.2152,Y -5.4648,Z 39,A -3.1094,B 0,C 0,E1 0.1598,E2 90.0711} C_DIS
LIN {X -4.6521,Y -5.9484,Z 39,A -3.1095,B 0,C 0,E1 0.1598,E2 90.0713} C_DIS
LIN {X -4.0469,Y -6.3782,Z 39,A -3.1056,B 0,C 0,E1 0.1598,E2 90.0713} C_DIS
LIN {X -3.4011,Y -6.7442,Z 39,A -3.0975,B 0,C 0,E1 0.1598,E2 90.0713} C_DIS
LIN {X -2.3996,Y -7.1671,Z 39,A -3.0787,B 0,C 0,E1 0.1598,E2 90.0713} C_DIS
LIN {X -1.1179,Y -7.4741,Z 39,A -3.0448,B 0,C 0,E1 0.1598,E2 90.0715} C_DIS
LIN {X 0.0049,Y -7.5548,Z 39,A -3.0071,B 0,C 0,E1 0.1598,E2 90.0715} C_DIS
Enddeposition()
LIN {X 0.0049,Y -7.5548,Z 39,A -3.0071,B 0,C 0,E1 0.1598,E2 90.0715} C_DIS
Startdeposition()
$VEL.CP = VEL_PRINT
LIN {X -0.6475,Y -8.4638,Z 39,A -3.0693,B 0,C 0,E1 0.1598,E2 90.0709} C_DIS
LIN {X -1.489,Y -8.3559,Z 39,A -3.0961,B 0,C 0,E1 0.1598,E2 90.0714} C_DIS
LIN {X -2.3158,Y -8.1655,Z 39,A -3.1183,B 0,C 0,E1 0.1598,E2 90.0714} C_DIS
LIN {X -3.4053,Y -7.7778,Z 39,A -3.1417,B 0,C 0,E1 0.1598,E2 90.0713} C_DIS
LIN {X -4.4691,Y -7.2186,Z 39,A -3.1569,B 0,C 0,E1 0.1598,E2 90.0712} C_DIS
LIN {X -5.3366,Y -6.5997,Z 39,A -3.1624,B 0,C 0,E1 0.1598,E2 90.0712} C_DIS
LIN {X -5.9718,Y -6.0311,Z 39,A -3.1616,B 0,C 0,E1 0.1598,E2 90.0712} C_DIS
LIN {X -6.5469,Y -5.4017,Z 39,A -3.156,B 0,C 0,E1 0.1598,E2 90.0712} C_DIS
LIN {X -7.0559,Y -4.7178,Z 39,A -3.1457,B 0,C 0,E1 0.1598,E2 90.0712} C_DIS
LIN {X -7.4937,Y -3.9862,Z 39,A -3.1307,B 0,C 0,E1 0.1598,E2 90.0712} C_DIS
LIN {X -7.8558,Y -3.2144,Z 39,A -3.1113,B 0,C 0,E1 0.1598,E2 90.0712} C_DIS
LIN {X -8.1386,Y -2.4101,Z 39,A -3.0877,B 0,C 0,E1 0.1598,E2 90.0712} C_DIS
LIN {X -8.3391,Y -1.5815,Z 39,A -3.06,B 0,C 0,E1 0.1598,E2 90.0712} C_DIS
LIN {X -8.4744,Y -0.5245,Z 39,A -3.0199,B 0,C 0,E1 0.1598,E2 90.0709} C_DIS
LIN {X -8.4647,Y 0.6692,Z 39,A -2.969,B 0,C 0,E1 0.1598,E2 90.0708} C_DIS
LIN {X -8.2966,Y 1.7888,Z 39,A -2.9157,B 0,C 0,E1 0.1598,E2 90.0711} C_DIS
LIN {X -7.9877,Y 2.8779,Z 39,A -2.8582,B 0,C 0,E1 0.1598,E2 90.0711} C_DIS
LIN {X -7.5287,Y 3.9188,Z 39,A -2.7974,B 0,C 0,E1 0.1598,E2 90.0713} C_DIS
LIN {X -7.1211,Y 4.6167,Z 39,A -2.7532,B 0,C 0,E1 0.1598,E2 90.0716} C_DIS
LIN {X -6.6491,Y 5.2728,Z 39,A -2.7081,B 0,C 0,E1 0.1598,E2 90.0717} C_DIS
LIN {X -5.8943,Y 6.1108,Z 39,A -2.6448,B 0,C 0,E1 0.1598,E2 90.0717} C_DIS
LIN {X -5.0793,Y 6.8002,Z 39,A -2.5857,B 0,C 0,E1 0.1598,E2 90.0719} C_DIS
LIN {X -4.3704,Y 7.2764,Z 39,A -2.5395,B 0,C 0,E1 0.1598,E2 90.0721} C_DIS
LIN {X -3.6171,Y 7.6788,Z 39,A -2.4947,B 0,C 0,E1 0.1598,E2 90.0721} C_DIS
LIN {X -2.8271,Y 8.0034,Z 39,A -2.4518,B 0,C 0,E1 0.1598,E2 90.0723} C_DIS
LIN {X -2.0085,Y 8.2468,Z 39,A -2.4113,B 0,C 0,E1 0.1598,E2 90.0723} C_DIS
LIN {X -1.1696,Y 8.4067,Z 39,A -2.3736,B 0,C 0,E1 0.1598,E2 90.0723} C_DIS
LIN {X -0.1054,Y 8.4903,Z 39,A -2.3308,B 0,C 0,E1 0.1598,E2 90.0725} C_DIS
LIN {X 1.0534,Y 8.4225,Z 39,A -2.2908,B 0,C 0,E1 0.1598,E2 90.0725} C_DIS
LIN {X 1.8969,Y 8.2727,Z 39,A -2.266,B 0,C 0,E1 0.1598,E2 90.0725} C_DIS
LIN {X 2.7212,Y 8.0393,Z 39,A -2.2455,B 0,C 0,E1 0.1598,E2 90.0725} C_DIS
LIN {X 3.5178,Y 7.724,Z 39,A -2.2294,B 0,C 0,E1 0.1598,E2 90.0725} C_DIS
LIN {X 4.5406,Y 7.1744,Z 39,A -2.2149,B 0,C 0,E1 0.1598,E2 90.0725} C_DIS
LIN {X 5.4966,Y 6.4705,Z 39,A -2.2094,B 0,C 0,E1 0.1598,E2 90.0723} C_DIS
LIN {X 6.264,Y 5.7271,Z 39,A -2.2128,B 0,C 0,E1 0.1598,E2 90.0723} C_DIS
LIN {X 6.8084,Y 5.0681,Z 39,A -2.2208,B 0,C 0,E1 0.1598,E2 90.0723} C_DIS
LIN {X 7.2838,Y 4.3576,Z 39,A -2.2335,B 0,C 0,E1 0.1598,E2 90.0723} C_DIS
LIN {X 7.6853,Y 3.6029,Z 39,A -2.2508,B 0,C 0,E1 0.1598,E2 90.0723} C_DIS
LIN {X 8.0084,Y 2.8116,Z 39,A -2.2726,B 0,C 0,E1 0.1598,E2 90.0722} C_DIS
LIN {X 8.2506,Y 1.9918,Z 39,A -2.2986,B 0,C 0,E1 0.1598,E2 90.0722} C_DIS
LIN {X 8.4091,Y 1.1518,Z 39,A -2.3286,B 0,C 0,E1 0.1598,E2 90.0721} C_DIS
LIN {X 8.4922,Y -0.0057,Z 39,A -2.3746,B 0,C 0,E1 0.1598,E2 90.0717} C_DIS
LIN {X 8.4112,Y -1.1697,Z 39,A -2.4272,B 0,C 0,E1 0.1598,E2 90.0716} C_DIS
LIN {X 8.1956,Y -2.2189,Z 39,A -2.4801,B 0,C 0,E1 0.1598,E2 90.0716} C_DIS
LIN {X 7.7816,Y -3.3872,Z 39,A -2.5449,B 0,C 0,E1 0.1598,E2 90.0714} C_DIS
LIN {X 7.3807,Y -4.1882,Z 39,A -2.5942,B 0,C 0,E1 0.1598,E2 90.0717} C_DIS
LIN {X 6.7354,Y -5.1687,Z 39,A -2.6597,B 0,C 0,E1 0.1598,E2 90.0716} C_DIS
LIN {X 6.0614,Y -5.94,Z 39,A -2.7175,B 0,C 0,E1 0.1598,E2 90.0716} C_DIS
LIN {X 5.46,Y -6.4966,Z 39,A -2.7634,B 0,C 0,E1 0.1598,E2 90.0717} C_DIS
LIN {X 4.8078,Y -6.9927,Z 39,A -2.8085,B 0,C 0,E1 0.1598,E2 90.0717} C_DIS
LIN {X 4.1109,Y -7.4236,Z 39,A -2.8525,B 0,C 0,E1 0.1598,E2 90.0717} C_DIS
LIN {X 3.3758,Y -7.7853,Z 39,A -2.8949,B 0,C 0,E1 0.1598,E2 90.0717} C_DIS
LIN {X 2.6092,Y -8.0744,Z 39,A -2.9353,B 0,C 0,E1 0.1598,E2 90.0717} C_DIS
LIN {X 1.8184,Y -8.2883,Z 39,A -2.9734,B 0,C 0,E1 0.1598,E2 90.0716} C_DIS
LIN {X 1.0106,Y -8.4252,Z 39,A -3.0089,B 0,C 0,E1 0.1598,E2 90.0716} C_DIS
LIN {X -0.0115,Y -8.4886,Z 39,A -3.049,B 0,C 0,E1 0.1598,E2 90.0716} C_DIS
Enddeposition()
LIN {X 0.0009,Y -4.7543,Z 40,A -2.875,B 0,C 0,E1 0.1598,E2 90.0604} C_DIS
Startdeposition()
$VEL.CP = VEL_PRINT
LIN {X 0.0009,Y -4.7543,Z 40,A -2.8807,B 0,C 0,E1 0.1598,E2 90.0661} C_DIS
LIN {X 0.8353,Y -4.6791,Z 40,A -2.8518,B 0,C 0,E1 0.1598,E2 90.0711} C_DIS
LIN {X 1.4852,Y -4.5144,Z 40,A -2.8216,B 0,C 0,E1 0.1598,E2 90.0718} C_DIS
LIN {X 2.105,Y -4.259,Z 40,A -2.788,B 0,C 0,E1 0.1598,E2 90.0718} C_DIS
LIN {X 2.6835,Y -3.9204,Z 40,A -2.7523,B 0,C 0,E1 0.1598,E2 90.0718} C_DIS
LIN {X 3.2086,Y -3.5038,Z 40,A -2.7153,B 0,C 0,E1 0.1598,E2 90.0718} C_DIS
LIN {X 3.6708,Y -3.0182,Z 40,A -2.6776,B 0,C 0,E1 0.1598,E2 90.0718} C_DIS
LIN {X 4.0596,Y -2.4719,Z 40,A -2.64,B 0,C 0,E1 0.1598,E2 90.0718} C_DIS
LIN {X 4.3646,Y -1.875,Z 40,A -2.6033,B 0,C 0,E1 0.1598,E2 90.0719} C_DIS
LIN {X 4.5854,Y -1.2423,Z 40,A -2.5682,B 0,C 0,E1 0.1598,E2 90.0719} C_DIS
LIN {X 4.7152,Y -0.5848,Z 40,A -2.5354,B 0,C 0,E1 0.1598,E2 90.0719} C_DIS
LIN {X 4.7494,Y 0.0847,Z 40,A -2.5056,B 0,C 0,E1 0.1598,E2 90.0719} C_DIS
LIN {X 4.6913,Y 0.7522,Z 40,A -2.4793,B 0,C 0,E1 0.1598,E2 90.072} C_DIS
LIN {X 4.5388,Y 1.4049,Z 40,A -2.4572,B 0,C 0,E1 0.1598,E2 90.072} C_DIS
LIN {X 4.297,Y 2.0302,Z 40,A -2.4395,B 0,C 0,E1 0.1598,E2 90.072} C_DIS
LIN {X 3.9681,Y 2.6144,Z 40,A -2.4267,B 0,C 0,E1 0.1598,E2 90.0721} C_DIS
LIN {X 3.5591,Y 3.1455,Z 40,A -2.4192,B 0,C 0,E1 0.1598,E2 90.0721} C_DIS
LIN {X 3.0811,Y 3.6152,Z 40,A -2.4169,B 0,C 0,E1 0.1598,E2 90.0722} C_DIS
LIN {X 2.543,Y 4.0149,Z 40,A -2.4198,B 0,C 0,E1 0.1598,E2 90.0722} C_DIS
LIN {X 1.8748,Y 4.3641,Z 40,A -2.4296,B 0,C 0,E1 0.1598,E2 90.0722} C_DIS
LIN {X 1.3227,Y 4.5618,Z 40,A -2.4416,B 0,C 0,E1 0.1598,E2 90.0722} C_DIS
LIN {X 0.668,Y 4.7049,Z 40,A -2.4597,B 0,C 0,E1 0.1598,E2 90.0722} C_DIS
LIN {X -0.0008,Y 4.7506,Z 40,A -2.4824,B 0,C 0,E1 0.1598,E2 90.0722} C_DIS
LIN {X -0.6693,Y 4.7033,Z 40,A -2.5091,B 0,C 0,E1 0.1598,E2 90.0722} C_DIS
LIN {X -1.3244,Y 4.5624,Z 40,A -2.5392,B 0,C 0,E1 0.1598,E2 90.0722} C_DIS
LIN {X -1.9534,Y 4.3307,Z 40,A -2.5722,B 0,C 0,E1 0.1598,E2 90.0722} C_DIS
LIN {X -2.5432,Y 4.0123,Z 40,A -2.6074,B 0,C 0,E1 0.1598,E2 90.072} C_DIS
LIN {X -3.0823,Y 3.6142,Z 40,A -2.6441,B 0,C 0,E1 0.1598,E2 90.072} C_DIS
LIN {X -3.5609,Y 3.145,Z 40,A -2.6815,B 0,C 0,E1 0.1598,E2 90.0719} C_DIS
LIN {X -3.9684,Y 2.6128,Z 40,A -2.719,B 0,C 0,E1 0.1598,E2 90.0719} C_DIS
LIN {X -4.2976,Y 2.0289,Z 40,A -2.7559,B 0,C 0,E1 0.1598,E2 90.0717} C_DIS
LIN {X -4.5408,Y 1.404,Z 40,A -2.7912,B 0,C 0,E1 0.1598,E2 90.0717} C_DIS
LIN {X -4.6932,Y 0.7511,Z 40,A -2.8245,B 0,C 0,E1 0.1598,E2 90.0716} C_DIS
LIN {X -4.7513,Y 0.0832,Z 40,A -2.8549,B 0,C 0,E1 0.1598,E2 90.0716} C_DIS
LIN {X -4.7159,Y -0.5862,Z 40,A -2.882,B 0,C 0,E1 0.1598,E2 90.0715} C_DIS
LIN {X -4.5611,Y -1.3242,Z 40,A -2.9075,B 0,C 0,E1 0.1598,E2 90.0715} C_DIS
LIN {X -4.3644,Y -1.8767,Z 40,A -2.9238,B 0,C 0,E1 0.1598,E2 90.0715} C_DIS
LIN {X -4.056,Y -2.4716,Z 40,A -2.9376,B 0,C 0,E1 0.1598,E2 90.0715} C_DIS
LIN {X -3.6698,Y -3.0196,Z 40,A -2.9467,B 0,C 0,E1 0.1598,E2 90.0715} C_DIS
LIN {X -3.2073,Y -3.5049,Z 40,A -2.9504,B 0,C 0,E1 0.1598,E2 90.0715} C_DIS
LIN {X -2.6821,Y -3.9213,Z 40,A -2.9488,B 0,C 0,E1 0.1598,E2 90.0715} C_DIS
LIN {X -2.1029,Y -4.2587,Z 40,A -2.9419,B 0,C 0,E1 0.1598,E2 90.0715} C_DIS
LIN {X -1.4832,Y -4.5136,Z 40,A -2.93,B 0,C 0,E1 0.1598,E2 90.0716} C_DIS
LIN {X -0.8333,Y -4.6775,Z 40,A -2.9131,B 0,C 0,E1 0.1598,E2 90.0716} C_DIS
LIN {X 0.0009,Y -4.7543,Z 40,A -2.8858,B 0,C 0,E1 0.1598,E2 90.0717} C_DIS
Enddeposition()
LIN {X 0.0009,Y -4.7543,Z 40,A -2.8858,B 0,C 0,E1 0.1598,E2 90.0717} C_DIS
Startdeposition()
$VEL.CP = VEL_PRINT
LIN {X -0.509,Y -5.6606,Z 40,A -2.9426,B 0,C 0,E1 0.1598,E2 90.0711} C_DIS
LIN {X -1.1976,Y -5.559,Z 40,A -2.9641,B 0,C 0,E1 0.1598,E2 90.0716} C_DIS
LIN {X -1.8673,Y -5.3688,Z 40,A -2.9806,B 0,C 0,E1 0.1598,E2 90.0716} C_DIS
LIN {X -2.5095,Y -5.1003,Z 40,A -2.9927,B 0,C 0,E1 0.1598,E2 90.0716} C_DIS
LIN {X -3.261,Y -4.662,Z 40,A -3.0016,B 0,C 0,E1 0.1598,E2 90.0714} C_DIS
LIN {X -3.8821,Y -4.1529,Z 40,A -3.0028,B 0,C 0,E1 0.1598,E2 90.0714} C_DIS
LIN {X -4.348,Y -3.6692,Z 40,A -2.9994,B 0,C 0,E1 0.1598,E2 90.0714} C_DIS
LIN {X -5.0513,Y -2.6093,Z 40,A -2.9798,B 0,C 0,E1 0.1598,E2 90.071} C_DIS
LIN {X -5.3691,Y -1.8661,Z 40,A -2.9603,B 0,C 0,E1 0.1598,E2 90.0713} C_DIS
LIN {X -5.5775,Y -1.0856,Z 40,A -2.9348,B 0,C 0,E1 0.1598,E2 90.0713} C_DIS
LIN {X -5.6768,Y -0.2838,Z 40,A -2.9045,B 0,C 0,E1 0.1598,E2 90.0713} C_DIS
LIN {X -5.6611,Y 0.5241,Z 40,A -2.8697,B 0,C 0,E1 0.1598,E2 90.0713} C_DIS
LIN {X -5.5271,Y 1.3209,Z 40,A -2.8311,B 0,C 0,E1 0.1598,E2 90.0715} C_DIS
LIN {X -5.2837,Y 2.0912,Z 40,A -2.7895,B 0,C 0,E1 0.1598,E2 90.0715} C_DIS
LIN {X -4.9336,Y 2.8191,Z 40,A -2.7459,B 0,C 0,E1 0.1598,E2 90.0716} C_DIS
LIN {X -4.4852,Y 3.4912,Z 40,A -2.7009,B 0,C 0,E1 0.1598,E2 90.0717} C_DIS
LIN {X -3.9461,Y 4.0933,Z 40,A -2.6556,B 0,C 0,E1 0.1598,E2 90.0718} C_DIS
LIN {X -3.3258,Y 4.6114,Z 40,A -2.6109,B 0,C 0,E1 0.1598,E2 90.072} C_DIS
LIN {X -2.4591,Y 5.1305,Z 40,A -2.5569,B 0,C 0,E1 0.1598,E2 90.072} C_DIS
LIN {X -1.3207,Y 5.5353,Z 40,A -2.4979,B 0,C 0,E1 0.1598,E2 90.0722} C_DIS
LIN {X -0.289,Y 5.677,Z 40,A -2.4539,B 0,C 0,E1 0.1598,E2 90.0722} C_DIS
LIN {X 0.5435,Y 5.6563,Z 40,A -2.4241,B 0,C 0,E1 0.1598,E2 90.0723} C_DIS
LIN {X 1.3649,Y 5.5177,Z 40,A -2.3996,B 0,C 0,E1 0.1598,E2 90.0723} C_DIS
LIN {X 2.1573,Y 5.2608,Z 40,A -2.3813,B 0,C 0,E1 0.1598,E2 90.0723} C_DIS
LIN {X 2.9025,Y 4.8882,Z 40,A -2.3696,B 0,C 0,E1 0.1598,E2 90.0723} C_DIS
LIN {X 3.5852,Y 4.4108,Z 40,A -2.3647,B 0,C 0,E1 0.1598,E2 90.0723} C_DIS
LIN {X 4.1914,Y 3.8395,Z 40,A -2.3666,B 0,C 0,E1 0.1598,E2 90.0723} C_DIS
LIN {X 4.7082,Y 3.1861,Z 40,A -2.3753,B 0,C 0,E1 0.1598,E2 90.0721} C_DIS
LIN {X 5.1233,Y 2.4637,Z 40,A -2.3907,B 0,C 0,E1 0.1598,E2 90.0721} C_DIS
LIN {X 5.4284,Y 1.6885,Z 40,A -2.4124,B 0,C 0,E1 0.1598,E2 90.0721} C_DIS
LIN {X 5.6166,Y 0.8769,Z 40,A -2.44,B 0,C 0,E1 0.1598,E2 90.0719} C_DIS
LIN {X 5.6851,Y 0.0467,Z 40,A -2.4728,B 0,C 0,E1 0.1598,E2 90.0719} C_DIS
LIN {X 5.6302,Y -0.7847,Z 40,A -2.5103,B 0,C 0,E1 0.1598,E2 90.0719} C_DIS
LIN {X 5.4543,Y -1.5989,Z 40,A -2.5515,B 0,C 0,E1 0.1598,E2 90.0719} C_DIS
LIN {X 5.1635,Y -2.3795,Z 40,A -2.5955,B 0,C 0,E1 0.1598,E2 90.0718} C_DIS
LIN {X 4.7604,Y -3.1086,Z 40,A -2.6414,B 0,C 0,E1 0.1598,E2 90.0718} C_DIS
LIN {X 4.2549,Y -3.771,Z 40,A -2.6882,B 0,C 0,E1 0.1598,E2 90.0718} C_DIS
LIN {X 3.6577,Y -4.352,Z 40,A -2.735,B 0,C 0,E1 0.1598,E2 90.0718} C_DIS
LIN {X 2.9821,Y -4.8395,Z 40,A -2.7806,B 0,C 0,E1 0.1598,E2 90.0718} C_DIS
LIN {X 2.2425,Y -5.2226,Z 40,A -2.8241,B 0,C 0,E1 0.1598,E2 90.0718} C_DIS
LIN {X 1.455,Y -5.4938,Z 40,A -2.8646,B 0,C 0,E1 0.1598,E2 90.0718} C_DIS
LIN {X 0.6363,Y -5.6467,Z 40,A -2.9011,B 0,C 0,E1 0.1598,E2 90.0717} C_DIS
LIN {X 0.0126,Y -5.6873,Z 40,A -2.9257,B 0,C 0,E1 0.1598,E2 90.0717} C_DIS
Enddeposition()
LIN {X 0.0126,Y -5.6873,Z 40,A -2.9257,B 0,C 0,E1 0.1598,E2 90.0717} C_DIS
Startdeposition()
$VEL.CP = VEL_PRINT
LIN {X 0.5592,Y -6.5949,Z 40,A -2.9439,B 0,C 0,E1 0.1598,E2 90.0711} C_DIS
LIN {X 1.297,Y -6.4906,Z 40,A -2.9129,B 0,C 0,E1 0.1598,E2 90.0717} C_DIS
LIN {X 2.0182,Y -6.3025,Z 40,A -2.8785,B 0,C 0,E1 0.1598,E2 90.0717} C_DIS
LIN {X 2.7141,Y -6.0357,Z 40,A -2.8416,B 0,C 0,E1 0.1598,E2 90.0717} C_DIS
LIN {X 3.3756,Y -5.6927,Z 40,A -2.8027,B 0,C 0,E1 0.1598,E2 90.0717} C_DIS
LIN {X 3.9942,Y -5.2769,Z 40,A -2.7622,B 0,C 0,E1 0.1598,E2 90.0718} C_DIS
LIN {X 4.5637,Y -4.7959,Z 40,A -2.7208,B 0,C 0,E1 0.1598,E2 90.0718} C_DIS
LIN {X 5.0738,Y -4.2525,Z 40,A -2.6789,B 0,C 0,E1 0.1598,E2 90.0718} C_DIS
LIN {X 5.5195,Y -3.6549,Z 40,A -2.637,B 0,C 0,E1 0.1598,E2 90.0718} C_DIS
LIN {X 5.8945,Y -3.0107,Z 40,A -2.5957,B 0,C 0,E1 0.1598,E2 90.0718} C_DIS
LIN {X 6.1969,Y -2.3294,Z 40,A -2.5555,B 0,C 0,E1 0.1598,E2 90.0719} C_DIS
LIN {X 6.4189,Y -1.6179,Z 40,A -2.517,B 0,C 0,E1 0.1598,E2 90.0719} C_DIS
LIN {X 6.5583,Y -0.8857,Z 40,A -2.4806,B 0,C 0,E1 0.1598,E2 90.0719} C_DIS
LIN {X 6.6159,Y -0.1427,Z 40,A -2.4468,B 0,C 0,E1 0.1598,E2 90.0719} C_DIS
LIN {X 6.5763,Y 0.7881,Z 40,A -2.4083,B 0,C 0,E1 0.1598,E2 90.0718} C_DIS
LIN {X 6.365,Y 1.8155,Z 40,A -2.3722,B 0,C 0,E1 0.1598,E2 90.0718} C_DIS
LIN {X 6.1302,Y 2.501,Z 40,A -2.352,B 0,C 0,E1 0.1598,E2 90.0721} C_DIS
LIN {X 5.821,Y 3.1564,Z 40,A -2.3355,B 0,C 0,E1 0.1598,E2 90.0721} C_DIS
LIN {X 5.438,Y 3.7715,Z 40,A -2.3235,B 0,C 0,E1 0.1598,E2 90.0722} C_DIS
LIN {X 4.9947,Y 4.3448,Z 40,A -2.3154,B 0,C 0,E1 0.1598,E2 90.0722} C_DIS
LIN {X 4.4891,Y 4.8639,Z 40,A -2.312,B 0,C 0,E1 0.1598,E2 90.0723} C_DIS
LIN {X 3.9309,Y 5.3259,Z 40,A -2.313,B 0,C 0,E1 0.1598,E2 90.0723} C_DIS
LIN {X 3.325,Y 5.7233,Z 40,A -2.3185,B 0,C 0,E1 0.1598,E2 90.0723} C_DIS
LIN {X 2.6792,Y 6.0519,Z 40,A -2.3284,B 0,C 0,E1 0.1598,E2 90.0723} C_DIS
LIN {X 2.0016,Y 6.3085,Z 40,A -2.3425,B 0,C 0,E1 0.1598,E2 90.0724} C_DIS
LIN {X 1.3002,Y 6.4908,Z 40,A -2.3606,B 0,C 0,E1 0.1598,E2 90.0724} C_DIS
LIN {X 0.5827,Y 6.5921,Z 40,A -2.3828,B 0,C 0,E1 0.1598,E2 90.0724} C_DIS
LIN {X -0.1414,Y 6.6176,Z 40,A -2.4085,B 0,C 0,E1 0.1598,E2 90.0724} C_DIS
LIN {X -0.8639,Y 6.5634,Z 40,A -2.4374,B 0,C 0,E1 0.1598,E2 90.0724} C_DIS
LIN {X -1.576,Y 6.4288,Z 40,A -2.4694,B 0,C 0,E1 0.1598,E2 90.0723} C_DIS
LIN {X -2.2693,Y 6.218,Z 40,A -2.5039,B 0,C 0,E1 0.1598,E2 90.0723} C_DIS
LIN {X -2.9354,Y 5.9327,Z 40,A -2.5405,B 0,C 0,E1 0.1598,E2 90.0721} C_DIS
LIN {X -3.567,Y 5.5774,Z 40,A -2.5788,B 0,C 0,E1 0.1598,E2 90.0721} C_DIS
LIN {X -4.1546,Y 5.1532,Z 40,A -2.6184,B 0,C 0,E1 0.1598,E2 90.072} C_DIS
LIN {X -4.693,Y 4.6681,Z 40,A -2.6588,B 0,C 0,E1 0.1598,E2 90.072} C_DIS
LIN {X -5.1751,Y 4.1271,Z 40,A -2.6994,B 0,C 0,E1 0.1598,E2 90.0718} C_DIS
LIN {X -5.7663,Y 3.2586,Z 40,A -2.7577,B 0,C 0,E1 0.1598,E2 90.0715} C_DIS
LIN {X -6.1464,Y 2.4599,Z 40,A -2.8055,B 0,C 0,E1 0.1598,E2 90.0715} C_DIS
LIN {X -6.3742,Y 1.7901,Z 40,A -2.8423,B 0,C 0,E1 0.1598,E2 90.0715} C_DIS
LIN {X -6.5289,Y 1.0996,Z 40,A -2.8772,B 0,C 0,E1 0.1598,E2 90.0715} C_DIS
LIN {X -6.6078,Y 0.3964,Z 40,A -2.9098,B 0,C 0,E1 0.1598,E2 90.0715} C_DIS
LIN {X -6.6126,Y -0.3111,Z 40,A -2.94,B 0,C 0,E1 0.1598,E2 90.0714} C_DIS
LIN {X -6.5436,Y -1.0153,Z 40,A -2.9672,B 0,C 0,E1 0.1598,E2 90.0714} C_DIS
LIN {X -6.3963,Y -1.7074,Z 40,A -2.9911,B 0,C 0,E1 0.1598,E2 90.0714} C_DIS
LIN {X -6.1755,Y -2.3797,Z 40,A -3.0115,B 0,C 0,E1 0.1598,E2 90.0714} C_DIS
LIN {X -5.8873,Y -3.0257,Z 40,A -3.0283,B 0,C 0,E1 0.1598,E2 90.0714} C_DIS
LIN {X -5.5307,Y -3.6369,Z 40,A -3.0411,B 0,C 0,E1 0.1598,E2 90.0714} C_DIS
LIN {X -5.1103,Y -4.2059,Z 40,A -3.0498,B 0,C 0,E1 0.1598,E2 90.0714} C_DIS
LIN {X -4.6323,Y -4.7275,Z 40,A -3.0544,B 0,C 0,E1 0.1598,E2 90.0714} C_DIS
LIN {X -4.1018,Y -5.1956,Z 40,A -3.0548,B 0,C 0,E1 0.1598,E2 90.0714} C_DIS
LIN {X -3.5249,Y -5.6053,Z 40,A -3.0511,B 0,C 0,E1 0.1598,E2 90.0714} C_DIS
LIN {X -2.9054,Y -5.9474,Z 40,A -3.0429,B 0,C 0,E1 0.1598,E2 90.0714} C_DIS
LIN {X -2.2536,Y -6.2224,Z 40,A -3.0307,B 0,C 0,E1 0.1598,E2 90.0714} C_DIS
LIN {X -1.5767,Y -6.4283,Z 40,A -3.0146,B 0,C 0,E1 0.1598,E2 90.0715} C_DIS
LIN {X -0.8817,Y -6.561,Z 40,A -2.9948,B 0,C 0,E1 0.1598,E2 90.0715} C_DIS
LIN {X 0.0006,Y -6.6222,Z 40,A -2.965,B 0,C 0,E1 0.1598,E2 90.0716} C_DIS
Enddeposition()
LIN {X 0.0006,Y -6.6222,Z 40,A -2.965,B 0,C 0,E1 0.1598,E2 90.0716} C_DIS
Startdeposition()
$VEL.CP = VEL_PRINT
LIN {X -0.4816,Y -7.5382,Z 40,A -3.0213,B 0,C 0,E1 0.1598,E2 90.071} C_DIS
LIN {X -1.4914,Y -7.4083,Z 40,A -3.0533,B 0,C 0,E1 0.1598,E2 90.0715} C_DIS
LIN {X -2.3938,Y -7.1689,Z 40,A -3.0762,B 0,C 0,E1 0.1598,E2 90.0715} C_DIS
LIN {X -3.3975,Y -6.7461,Z 40,A -3.095,B 0,C 0,E1 0.1598,E2 90.0713} C_DIS
LIN {X -4.044,Y -6.38,Z 40,A -3.1032,B 0,C 0,E1 0.1598,E2 90.0713} C_DIS
LIN {X -4.65,Y -5.9501,Z 40,A -3.1072,B 0,C 0,E1 0.1598,E2 90.0713} C_DIS
LIN {X -5.2132,Y -5.4657,Z 40,A -3.1072,B 0,C 0,E1 0.1598,E2 90.0713} C_DIS
LIN {X -5.9541,Y -4.6531,Z 40,A -3.0998,B 0,C 0,E1 0.1598,E2 90.0711} C_DIS
LIN {X -6.6344,Y -3.6175,Z 40,A -3.0807,B 0,C 0,E1 0.1598,E2 90.0709} C_DIS
LIN {X -7.0043,Y -2.8386,Z 40,A -3.0615,B 0,C 0,E1 0.1598,E2 90.0712} C_DIS
LIN {X -7.3509,Y -1.7376,Z 40,A -3.0273,B 0,C 0,E1 0.1598,E2 90.0709} C_DIS
LIN {X -7.4935,Y -0.9326,Z 40,A -2.9987,B 0,C 0,E1 0.1598,E2 90.0712} C_DIS
LIN {X -7.5526,Y -0.1171,Z 40,A -2.9664,B 0,C 0,E1 0.1598,E2 90.0712} C_DIS
LIN {X -7.5204,Y 0.7,Z 40,A -2.9307,B 0,C 0,E1 0.1598,E2 90.0713} C_DIS
LIN {X -7.2902,Y 1.991,Z 40,A -2.8671,B 0,C 0,E1 0.1598,E2 90.0709} C_DIS
LIN {X -6.7771,Y 3.3428,Z 40,A -2.7909,B 0,C 0,E1 0.1598,E2 90.0709} C_DIS
LIN {X -6.188,Y 4.3371,Z 40,A -2.7276,B 0,C 0,E1 0.1598,E2 90.0714} C_DIS
LIN {X -5.4823,Y 5.2003,Z 40,A -2.6652,B 0,C 0,E1 0.1598,E2 90.0716} C_DIS
LIN {X -4.6822,Y 5.9317,Z 40,A -2.6049,B 0,C 0,E1 0.1598,E2 90.0718} C_DIS
LIN {X -3.9551,Y 6.4388,Z 40,A -2.5567,B 0,C 0,E1 0.1598,E2 90.072} C_DIS
LIN {X -2.7517,Y 7.0327,Z 40,A -2.4872,B 0,C 0,E1 0.1598,E2 90.072} C_DIS
LIN {X -2.0152,Y 7.2787,Z 40,A -2.4497,B 0,C 0,E1 0.1598,E2 90.0723} C_DIS
LIN {X -1.2572,Y 7.4476,Z 40,A -2.4146,B 0,C 0,E1 0.1598,E2 90.0723} C_DIS
LIN {X -0.0777,Y 7.5571,Z 40,A -2.3665,B 0,C 0,E1 0.1598,E2 90.0724} C_DIS
LIN {X 1.1258,Y 7.4693,Z 40,A -2.3257,B 0,C 0,E1 0.1598,E2 90.0724} C_DIS
LIN {X 1.8438,Y 7.3286,Z 40,A -2.3052,B 0,C 0,E1 0.1598,E2 90.0724} C_DIS
LIN {X 2.8148,Y 7.0074,Z 40,A -2.283,B 0,C 0,E1 0.1598,E2 90.0724} C_DIS
LIN {X 3.7384,Y 6.5679,Z 40,A -2.2675,B 0,C 0,E1 0.1598,E2 90.0724} C_DIS
LIN {X 4.6568,Y 5.9467,Z 40,A -2.2599,B 0,C 0,E1 0.1598,E2 90.0724} C_DIS
LIN {X 5.3471,Y 5.3424,Z 40,A -2.2601,B 0,C 0,E1 0.1598,E2 90.0723} C_DIS
LIN {X 6.0706,Y 4.494,Z 40,A -2.2694,B 0,C 0,E1 0.1598,E2 90.0721} C_DIS
LIN {X 6.5024,Y 3.8432,Z 40,A -2.2814,B 0,C 0,E1 0.1598,E2 90.0723} C_DIS
LIN {X 6.8651,Y 3.1514,Z 40,A -2.2975,B 0,C 0,E1 0.1598,E2 90.0723} C_DIS
LIN {X 7.1533,Y 2.4255,Z 40,A -2.3177,B 0,C 0,E1 0.1598,E2 90.0722} C_DIS
LIN {X 7.41,Y 1.4835,Z 40,A -2.3482,B 0,C 0,E1 0.1598,E2 90.0718} C_DIS
LIN {X 7.5495,Y 0.2496,Z 40,A -2.3953,B 0,C 0,E1 0.1598,E2 90.0714} C_DIS
LIN {X 7.5417,Y -0.4794,Z 40,A -2.4272,B 0,C 0,E1 0.1598,E2 90.0719} C_DIS
LIN {X 7.4035,Y -1.5145,Z 40,A -2.4762,B 0,C 0,E1 0.1598,E2 90.0717} C_DIS
LIN {X 7.1234,Y -2.5234,Z 40,A -2.5296,B 0,C 0,E1 0.1598,E2 90.0717} C_DIS
LIN {X 6.7562,Y -3.3755,Z 40,A -2.5796,B 0,C 0,E1 0.1598,E2 90.0717} C_DIS
LIN {X 6.3938,Y -4.0232,Z 40,A -2.6207,B 0,C 0,E1 0.1598,E2 90.0718} C_DIS
LIN {X 5.7438,Y -4.9099,Z 40,A -2.6822,B 0,C 0,E1 0.1598,E2 90.0716} C_DIS
LIN {X 5.1305,Y -5.5486,Z 40,A -2.7321,B 0,C 0,E1 0.1598,E2 90.0716} C_DIS
LIN {X 4.3542,Y -6.1762,Z 40,A -2.7874,B 0,C 0,E1 0.1598,E2 90.0716} C_DIS
LIN {X 3.2271,Y -6.8332,Z 40,A -2.8568,B 0,C 0,E1 0.1598,E2 90.0716} C_DIS
LIN {X 2.2333,Y -7.2159,Z 40,A -2.9096,B 0,C 0,E1 0.1598,E2 90.0716} C_DIS
LIN {X 1.5582,Y -7.3919,Z 40,A -2.9419,B 0,C 0,E1 0.1598,E2 90.0716} C_DIS
LIN {X 0.8695,Y -7.503,Z 40,A -2.9719,B 0,C 0,E1 0.1598,E2 90.0716} C_DIS
LIN {X -0.001,Y -7.5548,Z 40,A -3.006,B 0,C 0,E1 0.1598,E2 90.0716} C_DIS
Enddeposition()
LIN {X -0.001,Y -7.5548,Z 40,A -3.006,B 0,C 0,E1 0.1598,E2 90.0716} C_DIS
Startdeposition()
$VEL.CP = VEL_PRINT
LIN {X 0.5263,Y -8.4698,Z 40,A -3.0253,B 0,C 0,E1 0.1598,E2 90.071} C_DIS
LIN {X 1.2485,Y -8.3943,Z 40,A -2.9961,B 0,C 0,E1 0.1598,E2 90.0715} C_DIS
LIN {X 2.392,Y -8.1477,Z 40,A -2.9437,B 0,C 0,E1 0.1598,E2 90.0716} C_DIS
LIN {X 3.4085,Y -7.7765,Z 40,A -2.8906,B 0,C 0,E1 0.1598,E2 90.0716} C_DIS
LIN {X 4.355,Y -7.2855,Z 40,A -2.8349,B 0,C 0,E1 0.1598,E2 90.0716} C_DIS
LIN {X 5.2355,Y -6.6839,Z 40,A -2.7769,B 0,C 0,E1 0.1598,E2 90.0716} C_DIS
LIN {X 6.0081,Y -6.0017,Z 40,A -2.7194,B 0,C 0,E1 0.1598,E2 90.0717} C_DIS
LIN {X 6.7074,Y -5.2051,Z 40,A -2.6597,B 0,C 0,E1 0.1598,E2 90.0717} C_DIS
LIN {X 7.3304,Y -4.277,Z 40,A -2.5971,B 0,C 0,E1 0.1598,E2 90.0717} C_DIS
LIN {X 7.8319,Y -3.2781,Z 40,A -2.5358,B 0,C 0,E1 0.1598,E2 90.0716} C_DIS
LIN {X 8.1773,Y -2.2893,Z 40,A -2.481,B 0,C 0,E1 0.1598,E2 90.0717} C_DIS
LIN {X 8.4202,Y -1.0721,Z 40,A -2.4198,B 0,C 0,E1 0.1598,E2 90.0715} C_DIS
LIN {X 8.4922,Y -0.0057,Z 40,A -2.3717,B 0,C 0,E1 0.1598,E2 90.0716} C_DIS
LIN {X 8.4102,Y 1.1442,Z 40,A -2.3256,B 0,C 0,E1 0.1598,E2 90.0716} C_DIS
LIN {X 8.2522,Y 1.9849,Z 40,A -2.2959,B 0,C 0,E1 0.1598,E2 90.0721} C_DIS
LIN {X 8.0104,Y 2.8053,Z 40,A -2.2699,B 0,C 0,E1 0.1598,E2 90.0721} C_DIS
LIN {X 7.6878,Y 3.5974,Z 40,A -2.248,B 0,C 0,E1 0.1598,E2 90.0721} C_DIS
LIN {X 7.2866,Y 4.3529,Z 40,A -2.2306,B 0,C 0,E1 0.1598,E2 90.0722} C_DIS
LIN {X 6.8114,Y 5.0641,Z 40,A -2.2179,B 0,C 0,E1 0.1598,E2 90.0723} C_DIS
LIN {X 6.2669,Y 5.7238,Z 40,A -2.2099,B 0,C 0,E1 0.1598,E2 90.0723} C_DIS
LIN {X 5.4995,Y 6.4681,Z 40,A -2.2064,B 0,C 0,E1 0.1598,E2 90.0723} C_DIS
LIN {X 4.536,Y 7.1772,Z 40,A -2.2119,B 0,C 0,E1 0.1598,E2 90.0723} C_DIS
LIN {X 3.5199,Y 7.7231,Z 40,A -2.2263,B 0,C 0,E1 0.1598,E2 90.0723} C_DIS
LIN {X 2.7229,Y 8.0388,Z 40,A -2.2424,B 0,C 0,E1 0.1598,E2 90.0725} C_DIS
LIN {X 1.8981,Y 8.2725,Z 40,A -2.263,B 0,C 0,E1 0.1598,E2 90.0725} C_DIS
LIN {X 1.0541,Y 8.4224,Z 40,A -2.2878,B 0,C 0,E1 0.1598,E2 90.0725} C_DIS
LIN {X -0.0971,Y 8.4905,Z 40,A -2.3275,B 0,C 0,E1 0.1598,E2 90.0725} C_DIS
LIN {X -1.1628,Y 8.4077,Z 40,A -2.3703,B 0,C 0,E1 0.1598,E2 90.0725} C_DIS
LIN {X -2.003,Y 8.2481,Z 40,A -2.4081,B 0,C 0,E1 0.1598,E2 90.0723} C_DIS
LIN {X -2.8229,Y 8.0049,Z 40,A -2.4487,B 0,C 0,E1 0.1598,E2 90.0723} C_DIS
LIN {X -3.6141,Y 7.6802,Z 40,A -2.4916,B 0,C 0,E1 0.1598,E2 90.0722} C_DIS
LIN {X -4.3685,Y 7.2775,Z 40,A -2.5364,B 0,C 0,E1 0.1598,E2 90.0722} C_DIS
LIN {X -5.0785,Y 6.8008,Z 40,A -2.5827,B 0,C 0,E1 0.1598,E2 90.072} C_DIS
LIN {X -5.9685,Y 6.0403,Z 40,A -2.6476,B 0,C 0,E1 0.1598,E2 90.0718} C_DIS
LIN {X -6.5678,Y 5.3748,Z 40,A -2.6978,B 0,C 0,E1 0.1598,E2 90.0718} C_DIS
LIN {X -7.2115,Y 4.4805,Z 40,A -2.7592,B 0,C 0,E1 0.1598,E2 90.0715} C_DIS
LIN {X -7.7945,Y 3.3662,Z 40,A -2.8275,B 0,C 0,E1 0.1598,E2 90.0712} C_DIS
LIN {X -8.1848,Y 2.2468,Z 40,A -2.8891,B 0,C 0,E1 0.1598,E2 90.071} C_DIS
LIN {X -8.4118,Y 1.1659,Z 40,A -2.9431,B 0,C 0,E1 0.1598,E2 90.071} C_DIS
LIN {X -8.4896,Y 0.1371,Z 40,A -2.9896,B 0,C 0,E1 0.1598,E2 90.071} C_DIS
LIN {X -8.438,Y -0.9423,Z 40,A -3.0333,B 0,C 0,E1 0.1598,E2 90.071} C_DIS
LIN {X -8.2507,Y -1.9919,Z 40,A -3.0709,B 0,C 0,E1 0.1598,E2 90.071} C_DIS
LIN {X -8.0093,Y -2.81,Z 40,A -3.0968,B 0,C 0,E1 0.1598,E2 90.071} C_DIS
LIN {X -7.6868,Y -3.5998,Z 40,A -3.1184,B 0,C 0,E1 0.1598,E2 90.071} C_DIS
LIN {X -7.2866,Y -4.353,Z 40,A -3.1356,B 0,C 0,E1 0.1598,E2 90.071} C_DIS
LIN {X -6.8127,Y -5.0623,Z 40,A -3.1483,B 0,C 0,E1 0.1598,E2 90.0711} C_DIS
LIN {X -6.2701,Y -5.7204,Z 40,A -3.1563,B 0,C 0,E1 0.1598,E2 90.0711} C_DIS
LIN {X -5.6641,Y -6.3208,Z 40,A -3.1595,B 0,C 0,E1 0.1598,E2 90.0711} C_DIS
LIN {X -5.0011,Y -6.8574,Z 40,A -3.158,B 0,C 0,E1 0.1598,E2 90.0712} C_DIS
LIN {X -3.9562,Y -7.5135,Z 40,A -3.1475,B 0,C 0,E1 0.1598,E2 90.0712} C_DIS
LIN {X -2.9237,Y -7.9709,Z 40,A -3.1292,B 0,C 0,E1 0.1598,E2 90.0712} C_DIS
LIN {X -1.9082,Y -8.2703,Z 40,A -3.1048,B 0,C 0,E1 0.1598,E2 90.0714} C_DIS
LIN {X -1.0743,Y -8.4194,Z 40,A -3.0806,B 0,C 0,E1 0.1598,E2 90.0714} C_DIS
LIN {X -0.018,Y -8.4887,Z 40,A -3.0448,B 0,C 0,E1 0.1598,E2 90.0715} C_DIS
Enddeposition()
LIN {X 0.0009,Y -4.7544,Z 41,A -2.8706,B 0,C 0,E1 0.1598,E2 90.0604} C_DIS
Startdeposition()
$VEL.CP = VEL_PRINT
LIN {X 0.0009,Y -4.7544,Z 41,A -2.8763,B 0,C 0,E1 0.1598,E2 90.0661} C_DIS
LIN {X -0.8333,Y -4.6776,Z 41,A -2.9086,B 0,C 0,E1 0.1598,E2 90.071} C_DIS
LIN {X -1.4832,Y -4.5137,Z 41,A -2.9261,B 0,C 0,E1 0.1598,E2 90.0716} C_DIS
LIN {X -2.1777,Y -4.2209,Z 41,A -2.9391,B 0,C 0,E1 0.1598,E2 90.0716} C_DIS
LIN {X -2.6822,Y -3.9215,Z 41,A -2.9449,B 0,C 0,E1 0.1598,E2 90.0716} C_DIS
LIN {X -3.2069,Y -3.5044,Z 41,A -2.9465,B 0,C 0,E1 0.1598,E2 90.0716} C_DIS
LIN {X -3.6697,Y -3.0195,Z 41,A -2.9428,B 0,C 0,E1 0.1598,E2 90.0716} C_DIS
LIN {X -4.056,Y -2.4716,Z 41,A -2.9338,B 0,C 0,E1 0.1598,E2 90.0715} C_DIS
LIN {X -4.3652,Y -1.877,Z 41,A -2.9199,B 0,C 0,E1 0.1598,E2 90.0715} C_DIS
LIN {X -4.5855,Y -1.2439,Z 41,A -2.9011,B 0,C 0,E1 0.1598,E2 90.0715} C_DIS
LIN {X -4.7166,Y -0.5864,Z 41,A -2.8781,B 0,C 0,E1 0.1598,E2 90.0715} C_DIS
LIN {X -4.7512,Y 0.0831,Z 41,A -2.851,B 0,C 0,E1 0.1598,E2 90.0715} C_DIS
LIN {X -4.6932,Y 0.7511,Z 41,A -2.8205,B 0,C 0,E1 0.1598,E2 90.0715} C_DIS
LIN {X -4.5408,Y 1.404,Z 41,A -2.7873,B 0,C 0,E1 0.1598,E2 90.0716} C_DIS
LIN {X -4.2977,Y 2.0288,Z 41,A -2.7519,B 0,C 0,E1 0.1598,E2 90.0716} C_DIS
LIN {X -3.9685,Y 2.6128,Z 41,A -2.715,B 0,C 0,E1 0.1598,E2 90.0718} C_DIS
LIN {X -3.5609,Y 3.145,Z 41,A -2.6775,B 0,C 0,E1 0.1598,E2 90.0718} C_DIS
LIN {X -3.0824,Y 3.6142,Z 41,A -2.64,B 0,C 0,E1 0.1598,E2 90.0719} C_DIS
LIN {X -2.5432,Y 4.0123,Z 41,A -2.6033,B 0,C 0,E1 0.1598,E2 90.072} C_DIS
LIN {X -1.9536,Y 4.331,Z 41,A -2.5681,B 0,C 0,E1 0.1598,E2 90.072} C_DIS
LIN {X -1.3245,Y 4.5621,Z 41,A -2.5352,B 0,C 0,E1 0.1598,E2 90.0722} C_DIS
LIN {X -0.6694,Y 4.7033,Z 41,A -2.505,B 0,C 0,E1 0.1598,E2 90.0722} C_DIS
LIN {X -0.0009,Y 4.7506,Z 41,A -2.4784,B 0,C 0,E1 0.1598,E2 90.0722} C_DIS
LIN {X 0.6678,Y 4.7048,Z 41,A -2.4557,B 0,C 0,E1 0.1598,E2 90.0722} C_DIS
LIN {X 1.3226,Y 4.5619,Z 41,A -2.4376,B 0,C 0,E1 0.1598,E2 90.0723} C_DIS
LIN {X 1.9514,Y 4.3303,Z 41,A -2.4243,B 0,C 0,E1 0.1598,E2 90.0723} C_DIS
LIN {X 2.5429,Y 4.0149,Z 41,A -2.4158,B 0,C 0,E1 0.1598,E2 90.0723} C_DIS
LIN {X 3.0809,Y 3.6151,Z 41,A -2.413,B 0,C 0,E1 0.1598,E2 90.0723} C_DIS
LIN {X 3.5591,Y 3.1456,Z 41,A -2.4153,B 0,C 0,E1 0.1598,E2 90.0723} C_DIS
LIN {X 3.9681,Y 2.6145,Z 41,A -2.4228,B 0,C 0,E1 0.1598,E2 90.0722} C_DIS
LIN {X 4.297,Y 2.0303,Z 41,A -2.4355,B 0,C 0,E1 0.1598,E2 90.0722} C_DIS
LIN {X 4.5389,Y 1.4051,Z 41,A -2.4532,B 0,C 0,E1 0.1598,E2 90.0721} C_DIS
LIN {X 4.6913,Y 0.7524,Z 41,A -2.4753,B 0,C 0,E1 0.1598,E2 90.0721} C_DIS
LIN {X 4.7494,Y 0.0848,Z 41,A -2.5016,B 0,C 0,E1 0.1598,E2 90.072} C_DIS
LIN {X 4.7152,Y -0.5846,Z 41,A -2.5314,B 0,C 0,E1 0.1598,E2 90.072} C_DIS
LIN {X 4.5854,Y -1.2422,Z 41,A -2.5642,B 0,C 0,E1 0.1598,E2 90.072} C_DIS
LIN {X 4.3647,Y -1.8749,Z 41,A -2.5993,B 0,C 0,E1 0.1598,E2 90.0719} C_DIS
LIN {X 4.0596,Y -2.4718,Z 41,A -2.6359,B 0,C 0,E1 0.1598,E2 90.0719} C_DIS
LIN {X 3.671,Y -3.0181,Z 41,A -2.6735,B 0,C 0,E1 0.1598,E2 90.0719} C_DIS
LIN {X 3.2075,Y -3.5024,Z 41,A -2.7112,B 0,C 0,E1 0.1598,E2 90.0719} C_DIS
LIN {X 2.6832,Y -3.9199,Z 41,A -2.7483,B 0,C 0,E1 0.1598,E2 90.0719} C_DIS
LIN {X 2.1054,Y -4.2595,Z 41,A -2.784,B 0,C 0,E1 0.1598,E2 90.0719} C_DIS
LIN {X 1.4852,Y -4.5143,Z 41,A -2.8176,B 0,C 0,E1 0.1598,E2 90.0718} C_DIS
LIN {X 0.8353,Y -4.6791,Z 41,A -2.8485,B 0,C 0,E1 0.1598,E2 90.0718} C_DIS
LIN {X 0.0009,Y -4.7544,Z 41,A -2.8823,B 0,C 0,E1 0.1598,E2 90.0718} C_DIS
Enddeposition()
LIN {X 0.0009,Y -4.7544,Z 41,A -2.8823,B 0,C 0,E1 0.1598,E2 90.0718} C_DIS
Startdeposition()
$VEL.CP = VEL_PRINT
LIN {X 0.2198,Y -5.6791,Z 41,A -2.9132,B 0,C 0,E1 0.1598,E2 90.0711} C_DIS
LIN {X 1.0409,Y -5.5865,Z 41,A -2.8796,B 0,C 0,E1 0.1598,E2 90.0717} C_DIS
LIN {X 1.8403,Y -5.3774,Z 41,A -2.8414,B 0,C 0,E1 0.1598,E2 90.0717} C_DIS
LIN {X 2.6011,Y -5.0546,Z 41,A -2.7997,B 0,C 0,E1 0.1598,E2 90.0717} C_DIS
LIN {X 3.3072,Y -4.6249,Z 41,A -2.7555,B 0,C 0,E1 0.1598,E2 90.0718} C_DIS
LIN {X 3.943,Y -4.0965,Z 41,A -2.7096,B 0,C 0,E1 0.1598,E2 90.0718} C_DIS
LIN {X 4.4939,Y -3.4802,Z 41,A -2.663,B 0,C 0,E1 0.1598,E2 90.0718} C_DIS
LIN {X 4.9523,Y -2.7923,Z 41,A -2.6168,B 0,C 0,E1 0.1598,E2 90.0718} C_DIS
LIN {X 5.3045,Y -2.0446,Z 41,A -2.5719,B 0,C 0,E1 0.1598,E2 90.0718} C_DIS
LIN {X 5.5463,Y -1.254,Z 41,A -2.5293,B 0,C 0,E1 0.1598,E2 90.0718} C_DIS
LIN {X 5.6678,Y -0.4363,Z 41,A -2.4899,B 0,C 0,E1 0.1598,E2 90.0718} C_DIS
LIN {X 5.6726,Y 0.3903,Z 41,A -2.4545,B 0,C 0,E1 0.1598,E2 90.0719} C_DIS
LIN {X 5.5553,Y 1.2085,Z 41,A -2.424,B 0,C 0,E1 0.1598,E2 90.0719} C_DIS
LIN {X 5.3195,Y 2.0008,Z 41,A -2.3989,B 0,C 0,E1 0.1598,E2 90.072} C_DIS
LIN {X 4.9739,Y 2.7514,Z 41,A -2.3797,B 0,C 0,E1 0.1598,E2 90.072} C_DIS
LIN {X 4.5214,Y 3.443,Z 41,A -2.367,B 0,C 0,E1 0.1598,E2 90.0721} C_DIS
LIN {X 3.9757,Y 4.0637,Z 41,A -2.3607,B 0,C 0,E1 0.1598,E2 90.0721} C_DIS
LIN {X 3.344,Y 4.5967,Z 41,A -2.3614,B 0,C 0,E1 0.1598,E2 90.0722} C_DIS
LIN {X 2.6416,Y 5.0321,Z 41,A -2.3689,B 0,C 0,E1 0.1598,E2 90.0722} C_DIS
LIN {X 1.8838,Y 5.3616,Z 41,A -2.3828,B 0,C 0,E1 0.1598,E2 90.0723} C_DIS
LIN {X 1.0866,Y 5.5785,Z 41,A -2.4031,B 0,C 0,E1 0.1598,E2 90.0723} C_DIS
LIN {X 0.2663,Y 5.6793,Z 41,A -2.4291,B 0,C 0,E1 0.1598,E2 90.0723} C_DIS
LIN {X -0.5602,Y 5.6588,Z 41,A -2.4604,B 0,C 0,E1 0.1598,E2 90.0723} C_DIS
LIN {X -1.1739,Y 5.5671,Z 41,A -2.4869,B 0,C 0,E1 0.1598,E2 90.0723} C_DIS
LIN {X -2.4007,Y 5.1588,Z 41,A -2.5494,B 0,C 0,E1 0.1598,E2 90.0721} C_DIS
LIN {X -3.3514,Y 4.5922,Z 41,A -2.6084,B 0,C 0,E1 0.1598,E2 90.0719} C_DIS
LIN {X -3.967,Y 4.0729,Z 41,A -2.6531,B 0,C 0,E1 0.1598,E2 90.0719} C_DIS
LIN {X -4.5017,Y 3.4708,Z 41,A -2.6982,B 0,C 0,E1 0.1598,E2 90.0718} C_DIS
LIN {X -4.9454,Y 2.799,Z 41,A -2.7429,B 0,C 0,E1 0.1598,E2 90.0717} C_DIS
LIN {X -5.2913,Y 2.0723,Z 41,A -2.7864,B 0,C 0,E1 0.1598,E2 90.0716} C_DIS
LIN {X -5.5312,Y 1.3039,Z 41,A -2.8277,B 0,C 0,E1 0.1598,E2 90.0715} C_DIS
LIN {X -5.6627,Y 0.5095,Z 41,A -2.8662,B 0,C 0,E1 0.1598,E2 90.0715} C_DIS
LIN {X -5.6764,Y -0.2955,Z 41,A -2.9007,B 0,C 0,E1 0.1598,E2 90.0714} C_DIS
LIN {X -5.5757,Y -1.0942,Z 41,A -2.9309,B 0,C 0,E1 0.1598,E2 90.0714} C_DIS
LIN {X -5.3671,Y -1.8717,Z 41,A -2.9562,B 0,C 0,E1 0.1598,E2 90.0714} C_DIS
LIN {X -5.0499,Y -2.6119,Z 41,A -2.9759,B 0,C 0,E1 0.1598,E2 90.0714} C_DIS
LIN {X -4.3466,Y -3.6708,Z 41,A -2.9946,B 0,C 0,E1 0.1598,E2 90.071} C_DIS
LIN {X -3.8804,Y -4.1545,Z 41,A -2.9985,B 0,C 0,E1 0.1598,E2 90.0714} C_DIS
LIN {X -3.2578,Y -4.6642,Z 41,A -2.9972,B 0,C 0,E1 0.1598,E2 90.0714} C_DIS
LIN {X -2.42,Y -5.1444,Z 41,A -2.9869,B 0,C 0,E1 0.1598,E2 90.0714} C_DIS
LIN {X -1.6992,Y -5.4224,Z 41,A -2.9724,B 0,C 0,E1 0.1598,E2 90.0716} C_DIS
LIN {X -0.9486,Y -5.6038,Z 41,A -2.9526,B 0,C 0,E1 0.1598,E2 90.0716} C_DIS
LIN {X 0.0131,Y -5.6874,Z 41,A -2.9209,B 0,C 0,E1 0.1598,E2 90.0716} C_DIS
Enddeposition()
LIN {X 0.0131,Y -5.6874,Z 41,A -2.9209,B 0,C 0,E1 0.1598,E2 90.0716} C_DIS
Startdeposition()
$VEL.CP = VEL_PRINT
LIN {X -0.53,Y -6.5988,Z 41,A -2.9791,B 0,C 0,E1 0.1598,E2 90.071} C_DIS
LIN {X -1.2317,Y -6.5045,Z 41,A -3.0014,B 0,C 0,E1 0.1598,E2 90.0715} C_DIS
LIN {X -1.9186,Y -6.3335,Z 41,A -3.0193,B 0,C 0,E1 0.1598,E2 90.0715} C_DIS
LIN {X -2.5844,Y -6.0933,Z 41,A -3.0335,B 0,C 0,E1 0.1598,E2 90.0715} C_DIS
LIN {X -3.221,Y -5.7838,Z 41,A -3.0437,B 0,C 0,E1 0.1598,E2 90.0715} C_DIS
LIN {X -3.8199,Y -5.4066,Z 41,A -3.0497,B 0,C 0,E1 0.1598,E2 90.0715} C_DIS
LIN {X -4.3749,Y -4.9673,Z 41,A -3.0514,B 0,C 0,E1 0.1598,E2 90.0714} C_DIS
LIN {X -4.8802,Y -4.4716,Z 41,A -3.0488,B 0,C 0,E1 0.1598,E2 90.0714} C_DIS
LIN {X -5.3298,Y -3.9248,Z 41,A -3.0421,B 0,C 0,E1 0.1598,E2 90.0714} C_DIS
LIN {X -5.719,Y -3.3336,Z 41,A -3.0313,B 0,C 0,E1 0.1598,E2 90.0714} C_DIS
LIN {X -6.0413,Y -2.7033,Z 41,A -3.0164,B 0,C 0,E1 0.1598,E2 90.0714} C_DIS
LIN {X -6.2952,Y -2.0427,Z 41,A -2.9978,B 0,C 0,E1 0.1598,E2 90.0714} C_DIS
LIN {X -6.4811,Y -1.3596,Z 41,A -2.9757,B 0,C 0,E1 0.1598,E2 90.0714} C_DIS
LIN {X -6.5883,Y -0.6598,Z 41,A -2.95,B 0,C 0,E1 0.1598,E2 90.0714} C_DIS
LIN {X -6.6188,Y 0.0474,Z 41,A -2.9211,B 0,C 0,E1 0.1598,E2 90.0714} C_DIS
LIN {X -6.578,Y 0.7541,Z 41,A -2.8897,B 0,C 0,E1 0.1598,E2 90.0714} C_DIS
LIN {X -6.4589,Y 1.4519,Z 41,A -2.8558,B 0,C 0,E1 0.1598,E2 90.0715} C_DIS
LIN {X -6.2675,Y 2.1334,Z 41,A -2.82,B 0,C 0,E1 0.1598,E2 90.0715} C_DIS
LIN {X -6.0037,Y 2.7903,Z 41,A -2.7825,B 0,C 0,E1 0.1598,E2 90.0716} C_DIS
LIN {X -5.4991,Y 3.6918,Z 41,A -2.7256,B 0,C 0,E1 0.1598,E2 90.0716} C_DIS
LIN {X -4.9408,Y 4.4045,Z 41,A -2.675,B 0,C 0,E1 0.1598,E2 90.0718} C_DIS
LIN {X -4.43,Y 4.918,Z 41,A -2.6345,B 0,C 0,E1 0.1598,E2 90.0719} C_DIS
LIN {X -3.8667,Y 5.3733,Z 41,A -2.5945,B 0,C 0,E1 0.1598,E2 90.072} C_DIS
LIN {X -3.2569,Y 5.7641,Z 41,A -2.5555,B 0,C 0,E1 0.1598,E2 90.072} C_DIS
LIN {X -2.6069,Y 6.0837,Z 41,A -2.518,B 0,C 0,E1 0.1598,E2 90.0722} C_DIS
LIN {X -1.9268,Y 6.3324,Z 41,A -2.4824,B 0,C 0,E1 0.1598,E2 90.0722} C_DIS
LIN {X -1.2236,Y 6.5055,Z 41,A -2.4492,B 0,C 0,E1 0.1598,E2 90.0722} C_DIS
LIN {X -0.5056,Y 6.601,Z 41,A -2.4186,B 0,C 0,E1 0.1598,E2 90.0723} C_DIS
LIN {X 0.2184,Y 6.6137,Z 41,A -2.3914,B 0,C 0,E1 0.1598,E2 90.0723} C_DIS
LIN {X 0.9399,Y 6.5522,Z 41,A -2.3674,B 0,C 0,E1 0.1598,E2 90.0724} C_DIS
LIN {X 1.65,Y 6.4098,Z 41,A -2.3472,B 0,C 0,E1 0.1598,E2 90.0724} C_DIS
LIN {X 2.3403,Y 6.1907,Z 41,A -2.331,B 0,C 0,E1 0.1598,E2 90.0724} C_DIS
Enddeposition()
END
